  MoveC 574 to (267.87, -55.04, -8.35) mm, rotated rx -180 ry 0 rz 0 deg; joints [19.602, -53.093, 148.442, 19.65, -94.169, 2.069] to (268.06, -55.49, -8.35) mm, rotated rx 180 ry 0 rz 0 deg; joints [19.58, -53.096, 148.465, 19.628, -94.189, 2.074]
  MoveL 575 to (268.06, -80.89, -8.35) mm, rotated rx 180 ry 0 rz 0 deg; joints [18.089, -53.148, 149.041, 18.147, -94.732, 2.105]
  MoveL 576 to (217.26, -80.89, -8.35) mm, rotated rx -180 ry 0 rz 0 deg; joints [17.156, -52.603, 145.594, 17.161, -91.988, 1.155]
  MoveL 577 to (217.26, -30.09, -8.35) mm, rotated rx -180 ry 0 rz 0 deg; joints [19.982, -52.424, 144.438, 19.979, -91.023, 0.96]
  MoveL 578 to (268.06, -30.09, -8.35) mm, rotated rx -180 ry 0 rz 0 deg; joints [21.044, -53.031, 147.845, 21.081, -93.623, 2.002]
  MoveL 579 to (268.06, -55.49, -8.35) mm, rotated rx 180 ry 0 rz 0 deg; joints [19.58, -53.096, 148.465, 19.628, -94.189, 2.074]
  MoveC 580 to (267.87, -55.94, -8.35) mm, rotated rx -180 ry 0 rz 0 deg; joints [19.55, -53.095, 148.464, 19.598, -94.189, 2.071] to (267.42, -56.12, -8.35) mm, rotated rx 180 ry 0 rz 0 deg; joints [19.53, -53.092, 148.438, 19.578, -94.169, 2.062]
  MoveL 581 to (266.79, -56.12, -8.35) mm, rotated rx 180 ry 0 rz 0 deg; joints [19.517, -53.086, 148.396, 19.564, -94.135, 2.048]
  MoveC 582 to (266.34, -56.12, -8.16) mm, rotated rx 180 ry 0 rz 0 deg; joints [19.508, -53.1, 148.369, 19.553, -94.096, 2.034] to (266.15, -56.12, -7.72) mm, rotated rx 180 ry 0 rz 0 deg; joints [19.504, -53.144, 148.364, 19.548, -94.051, 2.017]
  Set speed (1000.0 mm/s)
  MoveL 583 to (266.15, -56.12, 6) mm, rotated rx 180 ry 0 rz 0 deg; joints [19.495, -54.53, 148.591, 19.516, -92.959, 1.628]
  MoveL 584 to (139.15, -54.85, 6) mm, rotated rx 180 ry 0 rz 0 deg; joints [17.25, -52.506, 139.813, 17.276, -86.559, -0.527]
  Set speed (25.4 mm/s)
  MoveL 585 to (139.15, -54.85, -3.54) mm, rotated rx -180 ry 0 rz 0 deg; joints [17.254, -51.692, 139.679, 17.269, -87.209, -0.325]
  MoveC 586 to (139.34, -54.85, -3.99) mm, rotated rx 180 ry 0 rz 0 deg; joints [17.258, -51.657, 139.686, 17.272, -87.248, -0.313] to (139.79, -54.85, -4.17) mm, rotated rx 180 ry 0 rz 0 deg; joints [17.265, -51.649, 139.715, 17.279, -87.283, -0.302]
  Set speed (50.8 mm/s)
  MoveL 587 to (140.42, -54.85, -4.18) mm, rotated rx 180 ry 0 rz 0 deg; joints [17.275, -51.661, 139.76, 17.289, -87.315, -0.293]
  MoveC 588 to (140.87, -55.04, -4.17) mm, rotated rx -180 ry 0 rz 0 deg; joints [17.273, -51.67, 139.795, 17.286, -87.34, -0.285] to (141.06, -55.49, -4.17) mm, rotated rx -180 ry 0 rz 0 deg; joints [17.252, -51.676, 139.818, 17.265, -87.356, -0.279]
  MoveL 589 to (141.06, -80.89, -4.18) mm, rotated rx -180 ry 0 rz 0 deg; joints [15.918, -51.795, 140.349, 15.924, -87.74, -0.124]
  MoveL 590 to (90.26, -80.89, -4.17) mm, rotated rx 180 ry 0 rz 0 deg; joints [15.186, -50.797, 136.713, 15.235, -85.19, -0.8]
  MoveL 591 to (90.26, -30.09, -4.17) mm, rotated rx 180 ry 0 rz 0 deg; joints [17.729, -50.515, 135.638, 17.808, -84.486, -1.218]
  MoveL 592 to (141.06, -30.09, -4.17) mm, rotated rx -180 ry 0 rz 0 deg; joints [18.568, -51.543, 139.244, 18.589, -86.951, -0.46]
  MoveL 593 to (141.06, -55.49, -4.17) mm, rotated rx -180 ry 0 rz 0 deg; joints [17.252, -51.676, 139.818, 17.265, -87.356, -0.279]
  MoveC 594 to (140.87, -55.94, -4.18) mm, rotated rx 180 ry 0 rz 0 deg; joints [17.226, -51.675, 139.815, 17.239, -87.354, -0.279] to (140.42, -56.12, -4.17) mm, rotated rx -180 ry 0 rz 0 deg; joints [17.209, -51.668, 139.787, 17.222, -87.334, -0.284]
  MoveL 595 to (139.79, -56.12, -4.18) mm, rotated rx -180 ry 0 rz 0 deg; joints [17.199, -51.656, 139.742, 17.212, -87.303, -0.294]
  MoveC 596 to (139.34, -56.12, -3.99) mm, rotated rx -180 ry 0 rz 0 deg; joints [17.192, -51.663, 139.713, 17.205, -87.268, -0.304] to (139.15, -56.12, -3.54) mm, rotated rx -180 ry 0 rz 0 deg; joints [17.188, -51.698, 139.707, 17.203, -87.228, -0.317]
  Set speed (1000.0 mm/s)
  MoveL 597 to (139.15, -56.12, 5) mm, rotated rx 180 ry 0 rz 0 deg; joints [17.184, -52.427, 139.827, 17.208, -86.647, -0.497]
  MoveL 598 to (139.15, -54.85, 5) mm, rotated rx -180 ry 0 rz 0 deg; joints [17.25, -52.421, 139.8, 17.275, -86.628, -0.506]
  Set speed (25.4 mm/s)
  MoveL 599 to (139.15, -54.85, 1.83) mm, rotated rx -180 ry 0 rz 0 deg; joints [17.252, -52.15, 139.756, 17.273, -86.844, -0.438]
  MoveL 600 to (139.15, -54.85, -7.72) mm, rotated rx -180 ry 0 rz 0 deg; joints [17.257, -51.335, 139.618, 17.267, -87.49, -0.237]
  MoveC 601 to (139.34, -54.85, -8.16) mm, rotated rx -180 ry 0 rz 0 deg; joints [17.26, -51.3, 139.624, 17.27, -87.53, -0.225] to (139.79, -54.85, -8.35) mm, rotated rx -180 ry 0 rz 0 deg; joints [17.267, -51.293, 139.653, 17.277, -87.565, -0.215]
  Set speed (50.8 mm/s)
  MoveL 602 to (140.42, -54.85, -8.35) mm, rotated rx 180 ry 0 rz 0 deg; joints [17.277, -51.304, 139.698, 17.287, -87.596, -0.205]
  MoveC 603 to (140.87, -55.04, -8.35) mm, rotated rx 180 ry 0 rz 0 deg; joints [17.275, -51.313, 139.733, 17.284, -87.622, -0.197] to (141.06, -55.49, -8.35) mm, rotated rx -180 ry 0 rz 0 deg; joints [17.255, -51.319, 139.756, 17.264, -87.638, -0.191]
  MoveL 604 to (141.06, -80.89, -8.35) mm, rotated rx 180 ry 0 rz 0 deg; joints [15.92, -51.434, 140.287, 15.923, -88.027, -0.043]
  MoveL 605 to (90.26, -80.89, -8.35) mm, rotated rx -180 ry 0 rz 0 deg; joints [15.188, -50.458, 136.654, 15.231, -85.46, -0.726]
  MoveL 606 to (90.26, -30.09, -8.35) mm, rotated rx -180 ry 0 rz 0 deg; joints [17.731, -50.182, 135.58, 17.802, -84.747, -1.134]
  MoveL 607 to (141.06, -30.09, -8.35) mm, rotated rx 180 ry 0 rz 0 deg; joints [18.57, -51.189, 139.183, 18.587, -87.228, -0.367]
  MoveL 608 to (141.06, -55.49, -8.35) mm, rotated rx -180 ry 0 rz 0 deg; joints [17.255, -51.319, 139.756, 17.264, -87.638, -0.191]
  MoveC 609 to (140.87, -55.94, -8.35) mm, rotated rx 180 ry 0 rz 0 deg; joints [17.228, -51.318, 139.753, 17.237, -87.636, -0.191] to (140.42, -56.12, -8.35) mm, rotated rx 180 ry 0 rz 0 deg; joints [17.211, -51.31, 139.725, 17.22, -87.616, -0.197]
  MoveL 610 to (139.79, -56.12, -8.35) mm, rotated rx 180 ry 0 rz 0 deg; joints [17.201, -51.299, 139.681, 17.21, -87.585, -0.206]
  MoveC 611 to (139.34, -56.12, -8.16) mm, rotated rx -180 ry 0 rz 0 deg; joints [17.194, -51.306, 139.652, 17.204, -87.55, -0.217] to (139.15, -56.12, -7.72) mm, rotated rx 180 ry 0 rz 0 deg; joints [17.19, -51.341, 139.645, 17.201, -87.51, -0.229]
  Set speed (1000.0 mm/s)
  MoveL 612 to (139.15, -56.12, 6) mm, rotated rx -180 ry 0 rz 0 deg; joints [17.184, -52.513, 139.841, 17.209, -86.578, -0.518]
  MoveL 613 to (139.15, -235.88, 6) mm, rotated rx -180 ry 0 rz 0 deg; joints [7.413, -53.13, 142.645, 7.41, -88.649, 0.21]
  Set speed (25.4 mm/s)
  MoveL 614 to (139.15, -235.88, -3.54) mm, rotated rx -180 ry 0 rz 0 deg; joints [7.416, -52.274, 142.505, 7.412, -89.36, 0.302]
  MoveC 615 to (139.34, -235.88, -3.99) mm, rotated rx -180 ry 0 rz 0 deg; joints [7.418, -52.236, 142.511, 7.413, -89.403, 0.308] to (139.79, -235.88, -4.17) mm, rotated rx -180 ry 0 rz 0 deg; joints [7.421, -52.227, 142.541, 7.416, -89.442, 0.313]
  Set speed (50.8 mm/s)
  MoveL 616 to (140.42, -235.88, -4.18) mm, rotated rx -180 ry 0 rz 0 deg; joints [7.426, -52.238, 142.587, 7.421, -89.477, 0.317]
  MoveC 617 to (140.87, -236.07, -4.18) mm, rotated rx -180 ry 0 rz 0 deg; joints [7.419, -52.245, 142.621, 7.414, -89.503, 0.321] to (141.06, -236.52, -4.17) mm, rotated rx -180 ry 0 rz 0 deg; joints [7.395, -52.249, 142.639, 7.39, -89.517, 0.322]
  MoveL 618 to (141.06, -261.92, -4.18) mm, rotated rx 180 ry 0 rz 0 deg; joints [5.961, -52.283, 142.851, 5.956, -89.695, 0.331]
  MoveL 619 to (90.26, -261.92, -4.17) mm, rotated rx -180 ry 0 rz 0 deg; joints [5.676, -51.366, 139.142, 5.679, -86.918, 0.052]
  MoveL 620 to (90.26, -211.12, -4.18) mm, rotated rx -180 ry 0 rz 0 deg; joints [8.4, -51.27, 138.686, 8.41, -86.574, -0.106]
  MoveL 621 to (141.06, -211.12, -4.17) mm, rotated rx -180 ry 0 rz 0 deg; joints [8.819, -52.205, 142.38, 8.814, -89.304, 0.299]
  MoveL 622 to (141.06, -236.52, -4.17) mm, rotated rx -180 ry 0 rz 0 deg; joints [7.395, -52.249, 142.639, 7.39, -89.517, 0.322]
  MoveC 623 to (140.87, -236.97, -4.17) mm, rotated rx -180 ry 0 rz 0 deg; joints [7.368, -52.247, 142.629, 7.363, -89.51, 0.321] to (140.42, -237.15, -4.18) mm, rotated rx -180 ry 0 rz 0 deg; joints [7.354, -52.24, 142.599, 7.35, -89.486, 0.318]
  MoveL 624 to (139.79, -237.16, -4.17) mm, rotated rx 180 ry 0 rz 0 deg; joints [7.35, -52.229, 142.553, 7.345, -89.451, 0.314]
  MoveC 625 to (139.34, -237.16, -3.99) mm, rotated rx 180 ry 0 rz 0 deg; joints [7.346, -52.238, 142.523, 7.342, -89.413, 0.309] to (139.15, -237.15, -3.54) mm, rotated rx 180 ry 0 rz 0 deg; joints [7.345, -52.276, 142.517, 7.34, -89.369, 0.303]
  Set speed (1000.0 mm/s)
  MoveL 626 to (139.15, -237.15, 5) mm, rotated rx -180 ry 0 rz 0 deg; joints [7.342, -53.043, 142.643, 7.338, -88.734, 0.221]
  MoveL 627 to (139.15, -235.88, 5) mm, rotated rx 180 ry 0 rz 0 deg; joints [7.413, -53.041, 142.631, 7.41, -88.724, 0.219]
  Set speed (25.4 mm/s)
  MoveL 628 to (139.15, -235.88, 1.83) mm, rotated rx -180 ry 0 rz 0 deg; joints [7.414, -52.755, 142.585, 7.41, -88.961, 0.25]
  MoveL 629 to (139.15, -235.89, -7.72) mm, rotated rx -180 ry 0 rz 0 deg; joints [7.418, -51.899, 142.44, 7.413, -89.668, 0.342]
  MoveC 630 to (139.34, -235.88, -8.16) mm, rotated rx -180 ry 0 rz 0 deg; joints [7.419, -51.861, 142.447, 7.414, -89.711, 0.348] to (139.79, -235.88, -8.35) mm, rotated rx -180 ry 0 rz 0 deg; joints [7.423, -51.852, 142.476, 7.418, -89.75, 0.353]
  Set speed (50.8 mm/s)
  MoveL 631 to (140.42, -235.88, -8.35) mm, rotated rx -180 ry 0 rz 0 deg; joints [7.427, -51.862, 142.522, 7.422, -89.785, 0.358]
  MoveC 632 to (140.87, -236.07, -8.35) mm, rotated rx -180 ry 0 rz 0 deg; joints [7.42, -51.87, 142.556, 7.415, -89.811, 0.361] to (141.06, -236.52, -8.35) mm, rotated rx 180 ry 0 rz 0 deg; joints [7.396, -51.873, 142.574, 7.391, -89.825, 0.362]
  MoveL 633 to (141.06, -261.92, -8.35) mm, rotated rx 180 ry 0 rz 0 deg; joints [5.963, -51.906, 142.786, 5.958, -90.006, 0.364]
  MoveL 634 to (90.26, -261.92, -8.35) mm, rotated rx 180 ry 0 rz 0 deg; joints [5.677, -51.013, 139.081, 5.679, -87.208, 0.081]
  MoveL 635 to (90.26, -211.12, -8.35) mm, rotated rx -180 ry 0 rz 0 deg; joints [8.401, -50.92, 138.625, 8.409, -86.86, -0.063]
  MoveL 636 to (141.06, -211.12, -8.35) mm, rotated rx -180 ry 0 rz 0 deg; joints [8.821, -51.83, 142.316, 8.816, -89.61, 0.347]
  MoveL 637 to (141.06, -236.52, -8.35) mm, rotated rx 180 ry 0 rz 0 deg; joints [7.396, -51.873, 142.574, 7.391, -89.825, 0.362]
  MoveC 638 to (140.87, -236.97, -8.35) mm, rotated rx -180 ry 0 rz 0 deg; joints [7.37, -51.871, 142.564, 7.365, -89.818, 0.361] to (140.42, -237.16, -8.35) mm, rotated rx 180 ry 0 rz 0 deg; joints [7.356, -51.864, 142.534, 7.351, -89.795, 0.358]
  MoveL 639 to (139.79, -237.16, -8.35) mm, rotated rx -180 ry 0 rz 0 deg; joints [7.351, -51.854, 142.488, 7.346, -89.759, 0.353]
  MoveC 640 to (139.34, -237.15, -8.16) mm, rotated rx -180 ry 0 rz 0 deg; joints [7.348, -51.863, 142.458, 7.343, -89.721, 0.348] to (139.15, -237.15, -7.72) mm, rotated rx -180 ry 0 rz 0 deg; joints [7.346, -51.9, 142.452, 7.342, -89.678, 0.343]
  Set speed (1000.0 mm/s)
  MoveL 641 to (139.15, -237.15, 6) mm, rotated rx 180 ry 0 rz 0 deg; joints [7.341, -53.133, 142.657, 7.338, -88.659, 0.212]
  MoveL 642 to (266.15, -235.89, 6) mm, rotated rx -180 ry 0 rz 0 deg; joints [8.471, -54.806, 151.649, 8.512, -95.899, 1.283]
  Set speed (25.4 mm/s)
  MoveL 643 to (266.15, -235.89, -3.54) mm, rotated rx 180 ry 0 rz 0 deg; joints [8.476, -53.774, 151.483, 8.53, -96.755, 1.413]
  MoveC 644 to (266.34, -235.89, -3.99) mm, rotated rx -180 ry 0 rz 0 deg; joints [8.478, -53.727, 151.487, 8.533, -96.806, 1.421] to (266.79, -235.88, -4.17) mm, rotated rx -180 ry 0 rz 0 deg; joints [8.482, -53.709, 151.515, 8.538, -96.851, 1.428]
  Set speed (50.8 mm/s)
  MoveL 645 to (267.42, -235.89, -4.17) mm, rotated rx 180 ry 0 rz 0 deg; joints [8.488, -53.713, 151.559, 8.545, -96.89, 1.435]
  MoveC 646 to (267.87, -236.07, -4.18) mm, rotated rx 180 ry 0 rz 0 deg; joints [8.48, -53.715, 151.592, 8.538, -96.921, 1.438] to (268.06, -236.52, -4.17) mm, rotated rx -180 ry 0 rz 0 deg; joints [8.453, -53.716, 151.609, 8.511, -96.937, 1.437]
  MoveL 647 to (268.06, -261.92, -4.18) mm, rotated rx -180 ry 0 rz 0 deg; joints [6.819, -53.716, 151.842, 6.868, -97.198, 1.241]
  MoveL 648 to (217.26, -261.92, -4.18) mm, rotated rx 180 ry 0 rz 0 deg; joints [6.448, -53.314, 148.292, 6.459, -94.076, 0.832]
  MoveL 649 to (217.26, -211.12, -4.18) mm, rotated rx 180 ry 0 rz 0 deg; joints [9.532, -53.273, 147.796, 9.546, -93.591, 1.022]
  MoveL 650 to (268.06, -211.12, -4.17) mm, rotated rx -180 ry 0 rz 0 deg; joints [10.074, -53.712, 151.327, 10.138, -96.628, 1.609]
  MoveL 651 to (268.06, -236.52, -4.17) mm, rotated rx -180 ry 0 rz 0 deg; joints [8.453, -53.716, 151.609, 8.511, -96.937, 1.437]
  MoveC 652 to (267.87, -236.97, -4.17) mm, rotated rx -180 ry 0 rz 0 deg; joints [8.423, -53.715, 151.601, 8.48, -96.931, 1.432] to (267.42, -237.16, -4.17) mm, rotated rx -180 ry 0 rz 0 deg; joints [8.407, -53.713, 151.572, 8.463, -96.905, 1.426]
  MoveL 653 to (266.79, -237.15, -4.18) mm, rotated rx -180 ry 0 rz 0 deg; joints [8.401, -53.709, 151.528, 8.457, -96.865, 1.419]
  MoveC 654 to (266.34, -237.15, -3.99) mm, rotated rx -180 ry 0 rz 0 deg; joints [8.396, -53.727, 151.5, 8.451, -96.82, 1.412] to (266.15, -237.16, -3.54) mm, rotated rx -180 ry 0 rz 0 deg; joints [8.394, -53.774, 151.495, 8.449, -96.769, 1.404]
  Set speed (1000.0 mm/s)
  MoveL 655 to (266.15, -237.15, 5) mm, rotated rx 180 ry 0 rz 0 deg; joints [8.391, -54.698, 151.645, 8.432, -96.003, 1.289]
  MoveL 656 to (266.15, -235.89, 5) mm, rotated rx -180 ry 0 rz 0 deg; joints [8.472, -54.698, 151.632, 8.513, -95.989, 1.297]
  Set speed (25.4 mm/s)
  MoveL 657 to (266.15, -235.89, 1.83) mm, rotated rx -180 ry 0 rz 0 deg; joints [8.473, -54.354, 151.577, 8.52, -96.275, 1.34]
  MoveL 658 to (266.15, -235.89, -7.71) mm, rotated rx -180 ry 0 rz 0 deg; joints [8.477, -53.323, 151.406, 8.539, -97.125, 1.469]
  MoveC 659 to (266.34, -235.88, -8.16) mm, rotated rx -180 ry 0 rz 0 deg; joints [8.479, -53.276, 151.411, 8.542, -97.176, 1.477] to (266.79, -235.89, -8.35) mm, rotated rx -180 ry 0 rz 0 deg; joints [8.484, -53.258, 151.438, 8.547, -97.221, 1.484]
  Set speed (50.8 mm/s)
  MoveL 660 to (267.42, -235.89, -8.35) mm, rotated rx -180 ry 0 rz 0 deg; joints [8.49, -53.261, 151.482, 8.554, -97.261, 1.491]
  MoveC 661 to (267.87, -236.07, -8.35) mm, rotated rx 180 ry 0 rz 0 deg; joints [8.482, -53.264, 151.515, 8.547, -97.291, 1.495] to (268.06, -236.52, -8.35) mm, rotated rx -180 ry 0 rz 0 deg; joints [8.455, -53.264, 151.532, 8.52, -97.308, 1.493]
  MoveL 662 to (268.06, -261.92, -8.35) mm, rotated rx -180 ry 0 rz 0 deg; joints [6.82, -53.262, 151.764, 6.876, -97.573, 1.287]
  MoveL 663 to (217.26, -261.92, -8.35) mm, rotated rx 180 ry 0 rz 0 deg; joints [6.449, -52.894, 148.22, 6.464, -94.423, 0.871]
  MoveL 664 to (217.26, -211.12, -8.35) mm, rotated rx 180 ry 0 rz 0 deg; joints [9.534, -52.857, 147.725, 9.551, -93.931, 1.079]
  MoveL 665 to (268.06, -211.12, -8.35) mm, rotated rx -180 ry 0 rz 0 deg; joints [10.076, -53.263, 151.251, 10.147, -96.995, 1.675]
  MoveL 666 to (268.06, -236.52, -8.35) mm, rotated rx 180 ry 0 rz 0 deg; joints [8.455, -53.264, 151.532, 8.52, -97.308, 1.493]
  MoveC 667 to (267.87, -236.97, -8.35) mm, rotated rx -180 ry 0 rz 0 deg; joints [8.425, -53.264, 151.524, 8.489, -97.302, 1.488] to (267.42, -237.16, -8.35) mm, rotated rx 180 ry 0 rz 0 deg; joints [8.409, -53.261, 151.495, 8.472, -97.275, 1.481]
  MoveL 668 to (266.79, -237.16, -8.35) mm, rotated rx 180 ry 0 rz 0 deg; joints [8.403, -53.258, 151.451, 8.465, -97.235, 1.475]
  MoveC 669 to (266.34, -237.16, -8.16) mm, rotated rx -180 ry 0 rz 0 deg; joints [8.398, -53.276, 151.424, 8.46, -97.191, 1.467] to (266.15, -237.16, -7.72) mm, rotated rx 180 ry 0 rz 0 deg; joints [8.396, -53.323, 151.419, 8.457, -97.139, 1.459]
  Set speed (1000.0 mm/s)
  MoveL 670 to (266.15, -237.16, 6) mm, rotated rx 180 ry 0 rz 0 deg; joints [8.39, -54.806, 151.662, 8.43, -95.912, 1.275]
  MoveL 671 to (393.15, -235.88, 6) mm, rotated rx -180 ry 0 rz -30 deg; joints [-2.482, -54.877, 157.892, -33.089, -100.339, -6.392]
  Set speed (25.4 mm/s)
  MoveL 672 to (393.15, -235.89, -3.54) mm, rotated rx 180 ry 0 rz -30 deg; joints [-2.479, -53.673, 157.698, -33.192, -101.185, -6.954]
  MoveC 673 to (393.34, -235.88, -3.99) mm, rotated rx 180 ry 0 rz -30 deg; joints [-2.479, -53.615, 157.701, -33.199, -101.236, -6.988] to (393.79, -235.89, -4.18) mm, rotated rx 180 ry 0 rz -30 deg; joints [-2.481, -53.588, 157.727, -33.206, -101.28, -7.018]
  Set speed (50.8 mm/s)
  MoveL 674 to (394.42, -235.88, -4.18) mm, rotated rx -180 ry 0 rz -30 deg; joints [-2.483, -53.584, 157.77, -33.213, -101.319, -7.045]
  MoveC 675 to (394.87, -236.07, -4.18) mm, rotated rx 180 ry 0 rz -30 deg; joints [-2.498, -53.58, 157.8, -33.232, -101.345, -7.066] to (395.06, -236.52, -4.17) mm, rotated rx -180 ry 0 rz -30 deg; joints [-2.531, -53.579, 157.811, -33.266, -101.351, -7.08]
  MoveL 676 to (395.06, -261.92, -4.17) mm, rotated rx -180 ry 0 rz -30 deg; joints [-4.359, -53.578, 157.706, -35.101, -101.013, -7.398]
  MoveL 677 to (344.26, -261.92, -4.18) mm, rotated rx -180 ry 0 rz -30 deg; joints [-4.098, -53.729, 154.244, -34.491, -98.078, -5.261]
  MoveL 678 to (344.26, -211.12, -4.17) mm, rotated rx -180 ry 0 rz 0 deg; joints [11.013, -53.827, 156.503, 11.239, -101.571, 2.724]
  MoveL 679 to (395.06, -211.12, -4.18) mm, rotated rx -180 ry 0 rz 30 deg; joints [22.093, -54.031, 153.781, 52.376, -95.091, 7.51]
  MoveL 680 to (395.06, -236.52, -4.18) mm, rotated rx -180 ry 0 rz 30 deg; joints [20.495, -54.016, 154.413, 50.834, -95.712, 7.845]
  MoveC 681 to (394.87, -236.97, -4.17) mm, rotated rx -180 ry 0 rz 30 deg; joints [20.462, -54.015, 154.412, 50.802, -95.716, 7.841] to (394.42, -237.15, -4.18) mm, rotated rx -180 ry 0 rz 30 deg; joints [20.44, -54.015, 154.387, 50.777, -95.704, 7.82]
  MoveL 682 to (393.79, -237.15, -4.18) mm, rotated rx -180 ry 0 rz 30 deg; joints [20.425, -54.014, 154.346, 50.759, -95.681, 7.787]
  MoveC 683 to (393.34, -237.16, -3.99) mm, rotated rx 180 ry 0 rz 30 deg; joints [20.414, -54.035, 154.321, 50.745, -95.653, 7.749] to (393.15, -237.16, -3.54) mm, rotated rx 180 ry 0 rz 30 deg; joints [20.409, -54.086, 154.317, 50.736, -95.619, 7.706]
  Set speed (1000.0 mm/s)
  MoveL 684 to (393.15, -237.16, 5) mm, rotated rx -180 ry 0 rz 30 deg; joints [20.404, -55.074, 154.476, 50.67, -95.094, 7.061]
  MoveL 685 to (393.15, -235.88, 5) mm, rotated rx -180 ry 0 rz 30 deg; joints [20.484, -55.075, 154.445, 50.748, -95.065, 7.045]
  Set speed (25.4 mm/s)
  MoveL 686 to (393.15, -235.88, 1.82) mm, rotated rx 180 ry 0 rz 30 deg; joints [20.486, -54.707, 154.388, 50.772, -95.26, 7.286]
  MoveL 687 to (393.15, -235.88, -7.72) mm, rotated rx -180 ry 0 rz 30 deg; joints [20.493, -53.606, 154.206, 50.848, -95.84, 8.003]
  MoveC 688 to (393.34, -235.89, -8.16) mm, rotated rx -180 ry 0 rz 30 deg; joints [20.497, -53.554, 154.209, 50.857, -95.874, 8.046] to (393.79, -235.88, -8.35) mm, rotated rx 180 ry 0 rz 30 deg; joints [20.508, -53.533, 154.234, 50.871, -95.902, 8.084]
  Set speed (50.8 mm/s)
  MoveL 689 to (394.42, -235.89, -8.35) mm, rotated rx -180 ry 0 rz 30 deg; joints [20.523, -53.534, 154.275, 50.889, -95.925, 8.117]
  MoveC 690 to (394.87, -236.07, -8.35) mm, rotated rx -180 ry 0 rz 30 deg; joints [20.522, -53.534, 154.309, 50.891, -95.947, 8.143] to (395.06, -236.52, -8.35) mm, rotated rx -180 ry 0 rz 30 deg; joints [20.498, -53.533, 154.331, 50.869, -95.965, 8.158]
  MoveL 691 to (395.06, -261.92, -8.35) mm, rotated rx -180 ry 0 rz 30 deg; joints [18.866, -53.5, 154.914, 49.297, -96.601, 8.431]
  MoveL 692 to (344.26, -261.92, -8.35) mm, rotated rx 180 ry 0 rz 0 deg; joints [7.464, -53.229, 156.963, 7.649, -102.746, 2.083]
  MoveL 693 to (344.26, -211.12, -8.35) mm, rotated rx 180 ry 0 rz 0 deg; joints [11.015, -53.318, 156.416, 11.258, -101.985, 2.809]
  MoveL 694 to (395.06, -211.12, -8.35) mm, rotated rx -180 ry 0 rz 30 deg; joints [22.096, -53.555, 153.7, 52.407, -95.332, 7.825]
  MoveL 695 to (395.06, -236.52, -8.35) mm, rotated rx -180 ry 0 rz 30 deg; joints [20.498, -53.533, 154.331, 50.869, -95.965, 8.158]
  MoveC 696 to (394.87, -236.97, -8.35) mm, rotated rx 180 ry 0 rz 30 deg; joints [20.465, -53.533, 154.33, 50.836, -95.969, 8.154] to (394.42, -237.16, -8.35) mm, rotated rx -180 ry 0 rz 30 deg; joints [20.443, -53.532, 154.306, 50.812, -95.957, 8.132]
  MoveL 697 to (393.79, -237.15, -8.35) mm, rotated rx -180 ry 0 rz 30 deg; joints [20.428, -53.532, 154.265, 50.794, -95.934, 8.099]
  MoveC 698 to (393.34, -237.16, -8.16) mm, rotated rx 180 ry 0 rz 30 deg; joints [20.417, -53.553, 154.239, 50.779, -95.906, 8.061] to (393.15, -237.16, -7.72) mm, rotated rx -180 ry 0 rz 30 deg; joints [20.412, -53.605, 154.236, 50.77, -95.872, 8.018]
  Set speed (1000.0 mm/s)
  MoveL 699 to (393.15, -237.15, 6) mm, rotated rx -180 ry 0 rz 30 deg; joints [20.403, -55.19, 154.494, 50.663, -95.032, 6.985]
  MoveL 700 to (393.15, -422.22, 6) mm, rotated rx -180 ry 0 rz 30 deg; joints [7.885, -54.996, 157.593, 38.441, -99.031, 7.595]
  Set speed (25.4 mm/s)
  MoveL 701 to (393.15, -422.22, -3.54) mm, rotated rx -180 ry 0 rz 30 deg; joints [7.89, -53.801, 157.401, 38.549, -99.815, 8.228]
  MoveC 702 to (393.34, -422.22, -3.99) mm, rotated rx -180 ry 0 rz 30 deg; joints [7.892, -53.744, 157.404, 38.557, -99.862, 8.267] to (393.79, -422.22, -4.17) mm, rotated rx 180 ry 0 rz 30 deg; joints [7.896, -53.718, 157.43, 38.568, -99.902, 8.301]
  Set speed (50.8 mm/s)
  MoveL 703 to (394.42, -422.22, -4.18) mm, rotated rx -180 ry 0 rz 30 deg; joints [7.902, -53.714, 157.473, 38.579, -99.938, 8.331]
  MoveC 704 to (394.87, -422.41, -4.18) mm, rotated rx -180 ry 0 rz 30 deg; joints [7.894, -53.711, 157.505, 38.574, -99.966, 8.352] to (395.06, -422.86, -4.18) mm, rotated rx -180 ry 0 rz 30 deg; joints [7.863, -53.709, 157.522, 38.546, -99.985, 8.358]
  MoveL 705 to (395.06, -448.26, -4.17) mm, rotated rx -180 ry 0 rz 30 deg; joints [6.05, -53.668, 157.726, 36.75, -100.447, 8.159]
  MoveL 706 to (344.26, -448.26, -4.18) mm, rotated rx 180 ry 0 rz 30 deg; joints [5.687, -53.812, 154.272, 36.047, -97.596, 5.935]
  MoveL 707 to (344.26, -397.46, -4.18) mm, rotated rx 180 ry 0 rz 0 deg; joints [-2.223, -53.617, 157.457, -2.285, -102.959, -0.274]
  MoveL 708 to (395.06, -397.46, -4.18) mm, rotated rx -180 ry 0 rz -30 deg; joints [-13.884, -53.653, 156.233, -44.491, -98.421, -8.11]
  MoveL 709 to (395.06, -422.86, -4.17) mm, rotated rx 180 ry 0 rz -30 deg; joints [-15.601, -53.67, 155.791, -46.158, -97.837, -8.041]
  MoveC 710 to (394.87, -423.31, -4.18) mm, rotated rx -180 ry 0 rz -30 deg; joints [-15.628, -53.671, 155.77, -46.182, -97.819, -8.029] to (394.42, -423.49, -4.18) mm, rotated rx -180 ry 0 rz -30 deg; joints [-15.632, -53.672, 155.737, -46.183, -97.794, -8.005]
  MoveL 711 to (393.79, -423.49, -4.17) mm, rotated rx -180 ry 0 rz -30 deg; joints [-15.62, -53.673, 155.695, -46.167, -97.766, -7.971]
  MoveC 712 to (393.34, -423.49, -3.99) mm, rotated rx 180 ry 0 rz -30 deg; joints [-15.611, -53.696, 155.67, -46.153, -97.733, -7.935] to (393.15, -423.49, -3.54) mm, rotated rx -180 ry 0 rz -30 deg; joints [-15.608, -53.75, 155.666, -46.144, -97.694, -7.892]
  Set speed (1000.0 mm/s)
  MoveL 713 to (393.15, -423.49, 5) mm, rotated rx 180 ry 0 rz -30 deg; joints [-15.608, -54.772, 155.832, -46.065, -97.1, -7.27]
  MoveL 714 to (393.15, -422.22, 5) mm, rotated rx 180 ry 0 rz -30 deg; joints [-15.523, -54.772, 155.855, -45.982, -97.128, -7.276]
  Set speed (25.4 mm/s)
  MoveL 715 to (393.15, -422.22, 1.82) mm, rotated rx -180 ry 0 rz -30 deg; joints [-15.523, -54.392, 155.795, -46.011, -97.351, -7.508]
  MoveL 716 to (393.15, -422.22, -7.71) mm, rotated rx -180 ry 0 rz -30 deg; joints [-15.523, -53.251, 155.605, -46.103, -98.011, -8.198]
  MoveC 717 to (393.34, -422.22, -8.16) mm, rotated rx 180 ry 0 rz -30 deg; joints [-15.526, -53.197, 155.608, -46.112, -98.05, -8.24] to (393.79, -422.22, -8.35) mm, rotated rx -180 ry 0 rz -30 deg; joints [-15.534, -53.174, 155.634, -46.126, -98.082, -8.277]
  Set speed (50.8 mm/s)
  MoveL 718 to (394.42, -422.22, -8.35) mm, rotated rx 180 ry 0 rz -30 deg; joints [-15.546, -53.172, 155.676, -46.142, -98.111, -8.311]
  MoveC 719 to (394.87, -422.41, -8.35) mm, rotated rx 180 ry 0 rz -30 deg; joints [-15.567, -53.171, 155.702, -46.165, -98.127, -8.334] to (395.06, -422.86, -8.35) mm, rotated rx 180 ry 0 rz -30 deg; joints [-15.601, -53.17, 155.706, -46.199, -98.124, -8.342]
  MoveL 720 to (395.06, -448.26, -8.35) mm, rotated rx -180 ry 0 rz -30 deg; joints [-17.289, -53.19, 155.214, -47.832, -97.513, -8.212]
  MoveL 721 to (344.26, -448.26, -8.35) mm, rotated rx 180 ry 0 rz 0 deg; joints [-5.849, -53.098, 157.121, -6.009, -103.08, -1.181]
  MoveL 722 to (344.26, -397.46, -8.35) mm, rotated rx -180 ry 0 rz 0 deg; joints [-2.222, -53.096, 157.368, -2.288, -103.392, -0.292]
  MoveL 723 to (395.06, -397.46, -8.35) mm, rotated rx 180 ry 0 rz -30 deg; joints [-13.884, -53.148, 156.147, -44.535, -98.72, -8.407]
  MoveL 724 to (395.06, -422.86, -8.35) mm, rotated rx 180 ry 0 rz -30 deg; joints [-15.601, -53.17, 155.706, -46.199, -98.124, -8.342]
  MoveC 725 to (394.87, -423.31, -8.35) mm, rotated rx -180 ry 0 rz -30 deg; joints [-15.627, -53.171, 155.685, -46.224, -98.105, -8.331] to (394.42, -423.49, -8.35) mm, rotated rx -180 ry 0 rz -30 deg; joints [-15.631, -53.173, 155.652, -46.224, -98.081, -8.306]
  MoveL 726 to (393.79, -423.49, -8.35) mm, rotated rx -180 ry 0 rz -30 deg; joints [-15.62, -53.175, 155.61, -46.208, -98.052, -8.273]
  MoveC 727 to (393.34, -423.49, -8.16) mm, rotated rx 180 ry 0 rz -30 deg; joints [-15.611, -53.198, 155.585, -46.195, -98.02, -8.235] to (393.15, -423.49, -7.72) mm, rotated rx -180 ry 0 rz -30 deg; joints [-15.608, -53.252, 155.582, -46.185, -97.981, -8.193]
  Set speed (1000.0 mm/s)
  MoveL 728 to (393.15, -423.49, 6) mm, rotated rx -180 ry 0 rz -30 deg; joints [-15.608, -54.892, 155.851, -46.056, -97.03, -7.197]
  MoveL 729 to (266.15, -422.22, 6) mm, rotated rx 180 ry 0 rz 0 deg; joints [-3.642, -54.753, 152.184, -3.67, -96.547, -0.202]
  Set speed (25.4 mm/s)
  MoveL 730 to (266.15, -422.22, -3.54) mm, rotated rx 180 ry 0 rz 0 deg; joints [-3.64, -53.708, 152.015, -3.674, -97.421, -0.258]
  MoveC 731 to (266.34, -422.22, -3.99) mm, rotated rx 180 ry 0 rz 0 deg; joints [-3.64, -53.66, 152.02, -3.675, -97.474, -0.262] to (266.79, -422.22, -4.17) mm, rotated rx 180 ry 0 rz 0 deg; joints [-3.642, -53.642, 152.048, -3.678, -97.519, -0.265]
  Set speed (50.8 mm/s)
  MoveL 732 to (267.42, -422.22, -4.17) mm, rotated rx 180 ry 0 rz 0 deg; joints [-3.645, -53.645, 152.092, -3.681, -97.561, -0.268]
  MoveC 733 to (267.87, -422.41, -4.18) mm, rotated rx 180 ry 0 rz 0 deg; joints [-3.659, -53.647, 152.122, -3.695, -97.589, -0.272] to (268.06, -422.86, -4.18) mm, rotated rx -180 ry 0 rz 0 deg; joints [-3.689, -53.647, 152.133, -3.726, -97.599, -0.277]
  MoveL 734 to (268.06, -448.26, -4.18) mm, rotated rx 180 ry 0 rz 0 deg; joints [-5.343, -53.628, 151.992, -5.392, -97.458, -0.511]
  MoveL 735 to (217.26, -448.26, -4.17) mm, rotated rx -180 ry 0 rz 0 deg; joints [-5.051, -53.245, 148.437, -5.069, -94.302, -0.186]
  MoveL 736 to (217.26, -397.46, -4.18) mm, rotated rx -180 ry 0 rz 0 deg; joints [-1.917, -53.295, 148.659, -1.927, -94.491, 0.092]
  MoveL 737 to (268.06, -397.46, -4.17) mm, rotated rx -180 ry 0 rz 0 deg; joints [-2.029, -53.664, 152.223, -2.051, -97.684, -0.033]
  MoveL 738 to (268.06, -422.86, -4.18) mm, rotated rx -180 ry 0 rz 0 deg; joints [-3.689, -53.647, 152.133, -3.726, -97.599, -0.277]
  MoveC 739 to (267.87, -423.31, -4.18) mm, rotated rx 180 ry 0 rz 0 deg; joints [-3.718, -53.646, 152.118, -3.754, -97.585, -0.28] to (267.42, -423.49, -4.18) mm, rotated rx 180 ry 0 rz 0 deg; joints [-3.728, -53.644, 152.086, -3.764, -97.555, -0.28]
  MoveL 740 to (266.79, -423.49, -4.18) mm, rotated rx -180 ry 0 rz 0 deg; joints [-3.725, -53.641, 152.042, -3.761, -97.514, -0.277]
  MoveC 741 to (266.34, -423.49, -3.99) mm, rotated rx -180 ry 0 rz 0 deg; joints [-3.723, -53.659, 152.014, -3.759, -97.468, -0.274] to (266.15, -423.49, -3.54) mm, rotated rx -180 ry 0 rz 0 deg; joints [-3.723, -53.707, 152.009, -3.758, -97.415, -0.27]
  Set speed (1000.0 mm/s)
  MoveL 742 to (266.15, -423.49, 5) mm, rotated rx 180 ry 0 rz 0 deg; joints [-3.725, -54.642, 152.161, -3.753, -96.633, -0.219]
  MoveL 743 to (266.15, -422.22, 5) mm, rotated rx 180 ry 0 rz 0 deg; joints [-3.642, -54.643, 152.167, -3.67, -96.639, -0.208]
  Set speed (25.4 mm/s)
  MoveL 744 to (266.15, -422.22, 1.83) mm, rotated rx 180 ry 0 rz 0 deg; joints [-3.641, -54.295, 152.111, -3.672, -96.931, -0.227]
  MoveL 745 to (266.15, -422.22, -7.72) mm, rotated rx -180 ry 0 rz 0 deg; joints [-3.639, -53.252, 151.938, -3.677, -97.799, -0.283]
  MoveC 746 to (266.34, -422.22, -8.16) mm, rotated rx -180 ry 0 rz 0 deg; joints [-3.639, -53.204, 151.942, -3.678, -97.851, -0.286] to (266.79, -422.22, -8.35) mm, rotated rx 180 ry 0 rz 0 deg; joints [-3.641, -53.185, 151.97, -3.68, -97.897, -0.289]
  Set speed (50.8 mm/s)
  MoveL 747 to (267.42, -422.22, -8.35) mm, rotated rx 180 ry 0 rz 0 deg; joints [-3.644, -53.188, 152.014, -3.683, -97.939, -0.292]
  MoveC 748 to (267.87, -422.41, -8.35) mm, rotated rx -180 ry 0 rz 0 deg; joints [-3.658, -53.189, 152.044, -3.697, -97.967, -0.296] to (268.06, -422.86, -8.35) mm, rotated rx -180 ry 0 rz 0 deg; joints [-3.688, -53.19, 152.055, -3.728, -97.977, -0.302]
  MoveL 749 to (268.06, -448.26, -8.35) mm, rotated rx 180 ry 0 rz 0 deg; joints [-5.342, -53.172, 151.914, -5.396, -97.835, -0.547]
  MoveL 750 to (217.26, -448.26, -8.35) mm, rotated rx -180 ry 0 rz 0 deg; joints [-5.05, -52.823, 148.365, -5.07, -94.651, -0.217]
  MoveL 751 to (217.26, -397.46, -8.35) mm, rotated rx -180 ry 0 rz 0 deg; joints [-1.916, -52.872, 148.587, -1.927, -94.842, 0.08]
  MoveL 752 to (268.06, -397.46, -8.35) mm, rotated rx -180 ry 0 rz 0 deg; joints [-2.028, -53.206, 152.145, -2.052, -98.064, -0.047]
  MoveL 753 to (268.06, -422.86, -8.35) mm, rotated rx -180 ry 0 rz 0 deg; joints [-3.688, -53.19, 152.055, -3.728, -97.977, -0.302]
  MoveC 754 to (267.87, -423.31, -8.35) mm, rotated rx -180 ry 0 rz 0 deg; joints [-3.717, -53.189, 152.04, -3.756, -97.963, -0.305] to (267.42, -423.49, -8.35) mm, rotated rx -180 ry 0 rz 0 deg; joints [-3.727, -53.187, 152.008, -3.767, -97.933, -0.305]
  MoveL 755 to (266.79, -423.49, -8.35) mm, rotated rx 180 ry 0 rz 0 deg; joints [-3.724, -53.184, 151.964, -3.763, -97.892, -0.302]
  MoveC 756 to (266.34, -423.49, -8.16) mm, rotated rx 180 ry 0 rz 0 deg; joints [-3.722, -53.203, 151.936, -3.761, -97.846, -0.298] to (266.15, -423.49, -7.72) mm, rotated rx -180 ry 0 rz 0 deg; joints [-3.722, -53.251, 151.932, -3.76, -97.793, -0.295]
  Set speed (1000.0 mm/s)
  MoveL 757 to (266.15, -423.49, 6) mm, rotated rx -180 ry 0 rz 0 deg; joints [-3.725, -54.752, 152.178, -3.753, -96.541, -0.212]
  MoveL 758 to (139.15, -422.22, 6) mm, rotated rx -180 ry 0 rz 0 deg; joints [-3.182, -53.164, 143.134, -3.186, -89.101, 0.274]
  Set speed (25.4 mm/s)
  MoveL 759 to (139.15, -422.22, -3.54) mm, rotated rx -180 ry 0 rz 0 deg; joints [-3.18, -52.299, 142.992, -3.183, -89.823, 0.234]
  MoveC 760 to (139.34, -422.22, -3.99) mm, rotated rx -180 ry 0 rz 0 deg; joints [-3.18, -52.261, 142.999, -3.184, -89.867, 0.231] to (139.79, -422.22, -4.17) mm, rotated rx 180 ry 0 rz 0 deg; joints [-3.182, -52.252, 143.028, -3.185, -89.906, 0.229]
  Set speed (50.8 mm/s)
  MoveL 761 to (140.42, -422.22, -4.17) mm, rotated rx -180 ry 0 rz 0 deg; joints [-3.184, -52.262, 143.074, -3.187, -89.942, 0.227]
  MoveC 762 to (140.87, -422.41, -4.17) mm, rotated rx 180 ry 0 rz 0 deg; joints [-3.196, -52.269, 143.106, -3.199, -89.966, 0.226] to (141.06, -422.86, -4.17) mm, rotated rx 180 ry 0 rz 0 deg; joints [-3.222, -52.271, 143.118, -3.226, -89.976, 0.225]
  MoveL 763 to (141.06, -448.26, -4.18) mm, rotated rx 180 ry 0 rz 0 deg; joints [-4.668, -52.234, 142.989, -4.672, -89.883, 0.211]
  MoveL 764 to (90.26, -448.26, -4.18) mm, rotated rx -180 ry 0 rz 0 deg; joints [-4.443, -51.328, 139.277, -4.453, -87.086, 0.432]
  MoveL 765 to (90.26, -397.46, -4.18) mm, rotated rx -180 ry 0 rz 0 deg; joints [-1.686, -51.397, 139.481, -1.692, -87.215, 0.329]
  MoveL 766 to (141.06, -397.46, -4.18) mm, rotated rx -180 ry 0 rz 0 deg; joints [-1.771, -52.299, 143.2, -1.775, -90.031, 0.244]
  MoveL 767 to (141.06, -422.86, -4.17) mm, rotated rx 180 ry 0 rz 0 deg; joints [-3.222, -52.271, 143.118, -3.226, -89.976, 0.225]
  MoveC 768 to (140.87, -423.31, -4.18) mm, rotated rx 180 ry 0 rz 0 deg; joints [-3.247, -52.268, 143.102, -3.251, -89.964, 0.225] to (140.42, -423.49, -4.17) mm, rotated rx -180 ry 0 rz 0 deg; joints [-3.256, -52.26, 143.069, -3.26, -89.938, 0.226]
  MoveL 769 to (139.79, -423.49, -4.18) mm, rotated rx 180 ry 0 rz 0 deg; joints [-3.254, -52.25, 143.023, -3.258, -89.902, 0.228]
  MoveC 770 to (139.34, -423.49, -3.99) mm, rotated rx -180 ry 0 rz 0 deg; joints [-3.252, -52.26, 142.993, -3.256, -89.863, 0.231] to (139.15, -423.49, -3.54) mm, rotated rx 180 ry 0 rz 0 deg; joints [-3.252, -52.297, 142.987, -3.256, -89.819, 0.233]
  Set speed (1000.0 mm/s)
  MoveL 771 to (139.15, -423.49, 5) mm, rotated rx -180 ry 0 rz 0 deg; joints [-3.254, -53.071, 143.114, -3.258, -89.173, 0.27]
  MoveL 772 to (139.15, -422.22, 5) mm, rotated rx -180 ry 0 rz 0 deg; joints [-3.182, -53.073, 143.119, -3.186, -89.177, 0.27]
  Set speed (25.4 mm/s)
  MoveL 773 to (139.15, -422.22, 1.83) mm, rotated rx -180 ry 0 rz 0 deg; joints [-3.181, -52.785, 143.073, -3.185, -89.418, 0.256]
  MoveL 774 to (139.15, -422.22, -7.72) mm, rotated rx -180 ry 0 rz 0 deg; joints [-3.179, -51.92, 142.927, -3.183, -90.135, 0.216]
  MoveC 775 to (139.34, -422.22, -8.16) mm, rotated rx 180 ry 0 rz 0 deg; joints [-3.179, -51.883, 142.933, -3.183, -90.179, 0.214] to (139.79, -422.22, -8.35) mm, rotated rx -180 ry 0 rz 0 deg; joints [-3.181, -51.873, 142.963, -3.184, -90.219, 0.212]
  Set speed (50.8 mm/s)
  MoveL 776 to (140.42, -422.22, -8.35) mm, rotated rx -180 ry 0 rz 0 deg; joints [-3.183, -51.883, 143.009, -3.186, -90.255, 0.21]
  MoveC 777 to (140.87, -422.41, -8.35) mm, rotated rx 180 ry 0 rz 0 deg; joints [-3.195, -51.89, 143.041, -3.198, -90.28, 0.208] to (141.06, -422.86, -8.35) mm, rotated rx -180 ry 0 rz 0 deg; joints [-3.221, -51.892, 143.052, -3.225, -90.289, 0.207]
  MoveL 778 to (141.06, -448.26, -8.35) mm, rotated rx -180 ry 0 rz 0 deg; joints [-4.667, -51.856, 142.924, -4.671, -90.195, 0.185]
  MoveL 779 to (90.26, -448.26, -8.35) mm, rotated rx -180 ry 0 rz 0 deg; joints [-4.443, -50.973, 139.215, -4.451, -87.377, 0.409]
  MoveL 780 to (90.26, -397.46, -8.35) mm, rotated rx -180 ry 0 rz 0 deg; joints [-1.685, -51.042, 139.419, -1.69, -87.508, 0.32]
  MoveL 781 to (141.06, -397.46, -8.35) mm, rotated rx -180 ry 0 rz 0 deg; joints [-1.77, -51.919, 143.134, -1.774, -90.346, 0.235]
  MoveL 782 to (141.06, -422.86, -8.35) mm, rotated rx -180 ry 0 rz 0 deg; joints [-3.221, -51.892, 143.052, -3.225, -90.289, 0.207]
  MoveC 783 to (140.87, -423.31, -8.35) mm, rotated rx -180 ry 0 rz 0 deg; joints [-3.246, -51.888, 143.037, -3.25, -90.277, 0.207] to (140.42, -423.49, -8.35) mm, rotated rx -180 ry 0 rz 0 deg; joints [-3.255, -51.881, 143.004, -3.259, -90.251, 0.209]
  MoveL 784 to (139.79, -423.49, -8.35) mm, rotated rx -180 ry 0 rz 0 deg; joints [-3.253, -51.871, 142.958, -3.257, -90.215, 0.211]
  MoveC 785 to (139.34, -423.49, -8.16) mm, rotated rx 180 ry 0 rz 0 deg; joints [-3.252, -51.881, 142.928, -3.255, -90.176, 0.213] to (139.15, -423.49, -7.72) mm, rotated rx 180 ry 0 rz 0 deg; joints [-3.251, -51.919, 142.922, -3.255, -90.132, 0.215]
  Set speed (1000.0 mm/s)
  MoveL 786 to (139.15, -423.49, 6) mm, rotated rx 180 ry 0 rz 0 deg; joints [-3.254, -53.162, 143.129, -3.258, -89.097, 0.274]
  MoveL 787 to (-92.16, -422.22, 6) mm, rotated rx 180 ry 0 rz 0 deg; joints [-2.586, -47.662, 125.571, -2.657, -77.052, 0.829]
  Set speed (25.4 mm/s)
  MoveL 788 to (-92.16, -422.22, -3.54) mm, rotated rx -180 ry 0 rz 0 deg; joints [-2.584, -47.005, 125.456, -2.65, -77.594, 0.803]
  MoveC 789 to (-91.98, -422.22, -3.99) mm, rotated rx -180 ry 0 rz 0 deg; joints [-2.584, -46.979, 125.465, -2.65, -77.629, 0.801] to (-91.53, -422.22, -4.17) mm, rotated rx -180 ry 0 rz 0 deg; joints [-2.585, -46.979, 125.499, -2.65, -77.662, 0.8]
  Set speed (50.8 mm/s)
  MoveL 790 to (-90.89, -422.22, -4.18) mm, rotated rx 180 ry 0 rz 0 deg; joints [-2.587, -46.997, 125.549, -2.651, -77.695, 0.798]
  MoveC 791 to (-90.44, -422.41, -4.18) mm, rotated rx 180 ry 0 rz 0 deg; joints [-2.596, -47.009, 125.584, -2.661, -77.717, 0.799] to (-90.26, -422.86, -4.17) mm, rotated rx -180 ry 0 rz 0 deg; joints [-2.617, -47.014, 125.597, -2.683, -77.726, 0.803]
  MoveL 792 to (-90.26, -448.26, -4.17) mm, rotated rx -180 ry 0 rz 0 deg; joints [-3.794, -46.967, 125.483, -3.888, -77.672, 1.046]
  MoveL 793 to (-141.06, -448.26, -4.18) mm, rotated rx -180 ry 0 rz 0 deg; joints [-3.644, -45.471, 121.399, -3.775, -75.088, 1.19]
  MoveL 794 to (-141.06, -397.46, -4.17) mm, rotated rx -180 ry 0 rz 0 deg; joints [-1.381, -45.553, 121.584, -1.433, -75.165, 0.618]
  MoveL 795 to (-90.26, -397.46, -4.17) mm, rotated rx -180 ry 0 rz 0 deg; joints [-1.438, -47.047, 125.67, -1.476, -77.757, 0.563]
  MoveL 796 to (-90.26, -422.86, -4.17) mm, rotated rx -180 ry 0 rz 0 deg; joints [-2.617, -47.014, 125.597, -2.683, -77.726, 0.803]
  MoveC 797 to (-90.44, -423.31, -4.18) mm, rotated rx 180 ry 0 rz 0 deg; joints [-2.638, -47.008, 125.581, -2.704, -77.716, 0.808] to (-90.89, -423.49, -4.18) mm, rotated rx -180 ry 0 rz 0 deg; joints [-2.646, -46.995, 125.544, -2.712, -77.692, 0.811]
  MoveL 798 to (-91.53, -423.49, -4.18) mm, rotated rx 180 ry 0 rz 0 deg; joints [-2.644, -46.977, 125.494, -2.711, -77.66, 0.812]
  MoveC 799 to (-91.98, -423.49, -3.99) mm, rotated rx -180 ry 0 rz 0 deg; joints [-2.643, -46.977, 125.46, -2.71, -77.627, 0.813] to (-92.16, -423.49, -3.54) mm, rotated rx -180 ry 0 rz 0 deg; joints [-2.643, -47.003, 125.451, -2.71, -77.592, 0.815]
  Set speed (1000.0 mm/s)
  MoveL 800 to (-92.16, -423.49, 5) mm, rotated rx -180 ry 0 rz 0 deg; joints [-2.645, -47.591, 125.555, -2.717, -77.107, 0.839]
  MoveL 801 to (-92.16, -422.22, 5) mm, rotated rx -180 ry 0 rz 0 deg; joints [-2.586, -47.593, 125.559, -2.657, -77.109, 0.826]
  Set speed (25.4 mm/s)
  MoveL 802 to (-92.16, -422.22, 1.83) mm, rotated rx 180 ry 0 rz 0 deg; joints [-2.585, -47.374, 125.522, -2.654, -77.29, 0.817]
  MoveL 803 to (-92.16, -422.22, -7.71) mm, rotated rx -180 ry 0 rz 0 deg; joints [-2.583, -46.716, 125.403, -2.647, -77.829, 0.791]
  MoveC 804 to (-91.98, -422.22, -8.16) mm, rotated rx -180 ry 0 rz 0 deg; joints [-2.584, -46.691, 125.412, -2.647, -77.864, 0.79] to (-91.53, -422.22, -8.35) mm, rotated rx 180 ry 0 rz 0 deg; joints [-2.585, -46.69, 125.445, -2.647, -77.897, 0.788]
  Set speed (50.8 mm/s)
  MoveL 805 to (-90.89, -422.22, -8.35) mm, rotated rx -180 ry 0 rz 0 deg; joints [-2.586, -46.708, 125.496, -2.648, -77.93, 0.787]
  MoveC 806 to (-90.44, -422.41, -8.35) mm, rotated rx -180 ry 0 rz 0 deg; joints [-2.595, -46.721, 125.531, -2.658, -77.953, 0.788] to (-90.26, -422.86, -8.35) mm, rotated rx -180 ry 0 rz 0 deg; joints [-2.617, -46.725, 125.544, -2.679, -77.961, 0.792]
  MoveL 807 to (-90.26, -448.26, -8.35) mm, rotated rx -180 ry 0 rz 0 deg; joints [-3.794, -46.678, 125.43, -3.884, -77.907, 1.029]
  MoveL 808 to (-141.06, -448.26, -8.35) mm, rotated rx -180 ry 0 rz 0 deg; joints [-3.644, -45.197, 121.348, -3.771, -75.31, 1.174]
  MoveL 809 to (-141.06, -397.46, -8.35) mm, rotated rx -180 ry 0 rz 0 deg; joints [-1.381, -45.278, 121.532, -1.431, -75.389, 0.612]
  MoveL 810 to (-90.26, -397.46, -8.35) mm, rotated rx 180 ry 0 rz 0 deg; joints [-1.438, -46.758, 125.617, -1.474, -77.993, 0.557]
  MoveL 811 to (-90.26, -422.86, -8.35) mm, rotated rx -180 ry 0 rz 0 deg; joints [-2.617, -46.725, 125.544, -2.679, -77.961, 0.792]
  MoveC 812 to (-90.44, -423.31, -8.35) mm, rotated rx 180 ry 0 rz 0 deg; joints [-2.637, -46.719, 125.528, -2.7, -77.951, 0.796] to (-90.89, -423.49, -8.35) mm, rotated rx 180 ry 0 rz 0 deg; joints [-2.645, -46.706, 125.491, -2.709, -77.928, 0.799]
  MoveL 813 to (-91.53, -423.49, -8.35) mm, rotated rx -180 ry 0 rz 0 deg; joints [-2.643, -46.688, 125.441, -2.707, -77.895, 0.8]
  MoveC 814 to (-91.98, -423.49, -8.16) mm, rotated rx 180 ry 0 rz 0 deg; joints [-2.642, -46.689, 125.408, -2.707, -77.862, 0.802] to (-92.16, -423.49, -7.72) mm, rotated rx -180 ry 0 rz 0 deg; joints [-2.642, -46.714, 125.399, -2.707, -77.827, 0.803]
  Set speed (1000.0 mm/s)
  MoveL 815 to (-92.16, -423.49, 6) mm, rotated rx -180 ry 0 rz 0 deg; joints [-2.645, -47.66, 125.566, -2.718, -77.05, 0.842]
  MoveL 816 to (-219.16, -422.22, 6) mm, rotated rx -180 ry 0 rz 0 deg; joints [-2.345, -43.635, 115.134, -2.489, -70.646, 1.062]
  Set speed (25.4 mm/s)
  MoveL 817 to (-219.16, -422.22, -3.54) mm, rotated rx -180 ry 0 rz 0 deg; joints [-2.343, -43.053, 115.027, -2.48, -71.12, 1.04]
  MoveC 818 to (-218.98, -422.22, -3.99) mm, rotated rx -180 ry 0 rz 0 deg; joints [-2.343, -43.032, 115.038, -2.48, -71.152, 1.038] to (-218.53, -422.22, -4.17) mm, rotated rx -180 ry 0 rz 0 deg; joints [-2.344, -43.036, 115.074, -2.481, -71.184, 1.037]
  Set speed (50.8 mm/s)
  MoveL 819 to (-217.89, -422.22, -4.17) mm, rotated rx 180 ry 0 rz 0 deg; joints [-2.345, -43.057, 115.128, -2.481, -71.216, 1.036]
  MoveC 820 to (-217.44, -422.41, -4.17) mm, rotated rx -180 ry 0 rz 0 deg; joints [-2.354, -43.072, 115.165, -2.49, -71.239, 1.038] to (-217.26, -422.86, -4.18) mm, rotated rx 180 ry 0 rz 0 deg; joints [-2.373, -43.078, 115.179, -2.51, -71.248, 1.044]
  MoveL 821 to (-217.26, -448.26, -4.18) mm, rotated rx 180 ry 0 rz 0 deg; joints [-3.44, -43.028, 115.068, -3.638, -71.205, 1.394]
  MoveL 822 to (-268.06, -448.26, -4.17) mm, rotated rx -180 ry 0 rz 0 deg; joints [-3.317, -41.266, 110.69, -3.567, -68.59, 1.525]
  MoveL 823 to (-268.06, -397.46, -4.18) mm, rotated rx -180 ry 0 rz 0 deg; joints [-1.257, -41.351, 110.87, -1.353, -68.655, 0.746]
  MoveL 824 to (-217.26, -397.46, -4.17) mm, rotated rx 180 ry 0 rz 0 deg; joints [-1.304, -43.112, 115.25, -1.381, -71.273, 0.696]
  MoveL 825 to (-217.26, -422.86, -4.18) mm, rotated rx 180 ry 0 rz 0 deg; joints [-2.373, -43.078, 115.179, -2.51, -71.248, 1.044]
  MoveC 826 to (-217.44, -423.31, -4.17) mm, rotated rx 180 ry 0 rz 0 deg; joints [-2.391, -43.071, 115.162, -2.53, -71.238, 1.05] to (-217.89, -423.49, -4.17) mm, rotated rx -180 ry 0 rz 0 deg; joints [-2.399, -43.055, 115.123, -2.538, -71.215, 1.054]
  MoveL 827 to (-218.53, -423.49, -4.17) mm, rotated rx -180 ry 0 rz 0 deg; joints [-2.397, -43.034, 115.069, -2.537, -71.182, 1.055]
  MoveC 828 to (-218.98, -423.49, -3.99) mm, rotated rx 180 ry 0 rz 0 deg; joints [-2.397, -43.03, 115.033, -2.537, -71.15, 1.056] to (-219.16, -423.49, -3.54) mm, rotated rx 180 ry 0 rz 0 deg; joints [-2.396, -43.051, 115.023, -2.537, -71.118, 1.057]
  Set speed (1000.0 mm/s)
  MoveL 829 to (-219.16, -423.49, 5) mm, rotated rx 180 ry 0 rz 0 deg; joints [-2.398, -43.572, 115.119, -2.545, -70.695, 1.078]
  MoveL 830 to (-219.16, -422.22, 5) mm, rotated rx 180 ry 0 rz 0 deg; joints [-2.345, -43.574, 115.124, -2.488, -70.696, 1.06]
  Set speed (25.4 mm/s)
  MoveL 831 to (-219.16, -422.22, 1.82) mm, rotated rx -180 ry 0 rz 0 deg; joints [-2.344, -43.381, 115.088, -2.485, -70.854, 1.052]
  MoveL 832 to (-219.16, -422.22, -7.72) mm, rotated rx -180 ry 0 rz 0 deg; joints [-2.342, -42.798, 114.978, -2.477, -71.326, 1.03]
  MoveC 833 to (-218.98, -422.22, -8.16) mm, rotated rx 180 ry 0 rz 0 deg; joints [-2.343, -42.777, 114.988, -2.476, -71.357, 1.029] to (-218.53, -422.22, -8.35) mm, rotated rx -180 ry 0 rz 0 deg; joints [-2.343, -42.781, 115.024, -2.477, -71.389, 1.028]
  Set speed (50.8 mm/s)
  MoveL 834 to (-217.89, -422.22, -8.35) mm, rotated rx -180 ry 0 rz 0 deg; joints [-2.344, -42.802, 115.078, -2.477, -71.422, 1.026]
  MoveC 835 to (-217.44, -422.41, -8.35) mm, rotated rx -180 ry 0 rz 0 deg; joints [-2.353, -42.816, 115.115, -2.486, -71.445, 1.028] to (-217.26, -422.86, -8.35) mm, rotated rx -180 ry 0 rz 0 deg; joints [-2.372, -42.822, 115.13, -2.506, -71.454, 1.034]
  MoveL 836 to (-217.26, -448.26, -8.35) mm, rotated rx -180 ry 0 rz 0 deg; joints [-3.44, -42.773, 115.019, -3.633, -71.41, 1.38]
  MoveL 837 to (-268.06, -448.26, -8.35) mm, rotated rx -180 ry 0 rz 0 deg; joints [-3.316, -41.022, 110.641, -3.561, -68.786, 1.512]
  MoveL 838 to (-268.06, -397.46, -8.35) mm, rotated rx 180 ry 0 rz 0 deg; joints [-1.256, -41.106, 110.821, -1.351, -68.851, 0.741]
  MoveL 839 to (-217.26, -397.46, -8.35) mm, rotated rx -180 ry 0 rz 0 deg; joints [-1.303, -42.856, 115.2, -1.378, -71.48, 0.69]
  MoveL 840 to (-217.26, -422.86, -8.35) mm, rotated rx -180 ry 0 rz 0 deg; joints [-2.372, -42.822, 115.13, -2.506, -71.454, 1.034]
  MoveC 841 to (-217.44, -423.31, -8.35) mm, rotated rx -180 ry 0 rz 0 deg; joints [-2.391, -42.815, 115.112, -2.526, -71.444, 1.04] to (-217.89, -423.49, -8.35) mm, rotated rx -180 ry 0 rz 0 deg; joints [-2.398, -42.8, 115.073, -2.534, -71.42, 1.044]
  MoveL 842 to (-218.53, -423.49, -8.35) mm, rotated rx -180 ry 0 rz 0 deg; joints [-2.397, -42.778, 115.02, -2.533, -71.388, 1.045]
  MoveC 843 to (-218.98, -423.49, -8.16) mm, rotated rx -180 ry 0 rz 0 deg; joints [-2.396, -42.775, 114.984, -2.533, -71.355, 1.046] to (-219.16, -423.49, -7.72) mm, rotated rx 180 ry 0 rz 0 deg; joints [-2.396, -42.796, 114.973, -2.533, -71.324, 1.047]
  Set speed (1000.0 mm/s)
  MoveL 844 to (-219.16, -423.49, 6) mm, rotated rx 180 ry 0 rz 0 deg; joints [-2.398, -43.633, 115.13, -2.546, -70.645, 1.08]
  MoveL 845 to (-346.16, -422.22, 6) mm, rotated rx 180 ry 0 rz 0 deg; joints [-2.145, -38.951, 103.885, -2.389, -64.084, 1.284]
  Set speed (25.4 mm/s)
  MoveL 846 to (-346.16, -422.22, -3.54) mm, rotated rx -180 ry 0 rz 0 deg; joints [-2.143, -38.428, 103.781, -2.379, -64.502, 1.264]
  MoveC 847 to (-345.98, -422.22, -3.99) mm, rotated rx 180 ry 0 rz 0 deg; joints [-2.143, -38.41, 103.793, -2.378, -64.532, 1.263] to (-345.53, -422.22, -4.17) mm, rotated rx 180 ry 0 rz 0 deg; joints [-2.144, -38.418, 103.833, -2.378, -64.564, 1.262]
  Set speed (50.8 mm/s)
  MoveL 848 to (-344.89, -422.22, -4.18) mm, rotated rx -180 ry 0 rz 0 deg; joints [-2.145, -38.443, 103.891, -2.379, -64.598, 1.261]
  MoveC 849 to (-344.44, -422.41, -4.17) mm, rotated rx -180 ry 0 rz 0 deg; joints [-2.153, -38.46, 103.932, -2.387, -64.621, 1.263] to (-344.26, -422.86, -4.18) mm, rotated rx -180 ry 0 rz 0 deg; joints [-2.17, -38.466, 103.948, -2.406, -64.631, 1.271]
  MoveL 850 to (-344.26, -448.26, -4.17) mm, rotated rx 180 ry 0 rz 0 deg; joints [-3.147, -38.414, 103.837, -3.488, -64.593, 1.723]
  MoveL 851 to (-395.06, -448.26, -4.17) mm, rotated rx 180 ry 0 rz 0 deg; joints [-3.043, -36.363, 99.045, -3.456, -61.854, 1.858]
  MoveL 852 to (-395.06, -397.46, -4.18) mm, rotated rx -180 ry 0 rz 0 deg; joints [-1.153, -36.452, 99.227, -1.311, -61.911, 0.872]
  MoveL 853 to (-344.26, -397.46, -4.18) mm, rotated rx -180 ry 0 rz 0 deg; joints [-1.192, -38.502, 104.018, -1.323, -64.653, 0.821]
  MoveL 854 to (-344.26, -422.86, -4.18) mm, rotated rx -180 ry 0 rz 0 deg; joints [-2.17, -38.466, 103.948, -2.406, -64.631, 1.271]
  MoveC 855 to (-344.44, -423.31, -4.17) mm, rotated rx 180 ry 0 rz 0 deg; joints [-2.187, -38.458, 103.929, -2.425, -64.62, 1.279] to (-344.89, -423.49, -4.18) mm, rotated rx -180 ry 0 rz 0 deg; joints [-2.194, -38.44, 103.887, -2.433, -64.596, 1.283]
  MoveL 856 to (-345.53, -423.49, -4.18) mm, rotated rx -180 ry 0 rz 0 deg; joints [-2.193, -38.416, 103.828, -2.432, -64.562, 1.284]
  MoveC 857 to (-345.98, -423.49, -3.99) mm, rotated rx -180 ry 0 rz 0 deg; joints [-2.192, -38.408, 103.789, -2.432, -64.53, 1.286] to (-346.16, -423.49, -3.54) mm, rotated rx -180 ry 0 rz 0 deg; joints [-2.192, -38.426, 103.776, -2.433, -64.501, 1.287]
  Set speed (1000.0 mm/s)
  MoveL 858 to (-346.16, -423.49, 5) mm, rotated rx -180 ry 0 rz 0 deg; joints [-2.193, -38.894, 103.87, -2.442, -64.126, 1.305]
  MoveL 859 to (-346.16, -422.22, 5) mm, rotated rx 180 ry 0 rz 0 deg; joints [-2.144, -38.896, 103.874, -2.388, -64.128, 1.282]
  Set speed (25.4 mm/s)
  MoveL 860 to (-346.16, -422.22, 1.82) mm, rotated rx 180 ry 0 rz 0 deg; joints [-2.144, -38.722, 103.84, -2.384, -64.267, 1.275]
  MoveL 861 to (-346.16, -422.22, -7.71) mm, rotated rx -180 ry 0 rz 0 deg; joints [-2.142, -38.198, 103.733, -2.374, -64.684, 1.256]
  MoveC 862 to (-345.98, -422.22, -8.16) mm, rotated rx -180 ry 0 rz 0 deg; joints [-2.143, -38.181, 103.745, -2.374, -64.714, 1.254] to (-345.53, -422.22, -8.35) mm, rotated rx -180 ry 0 rz 0 deg; joints [-2.143, -38.188, 103.785, -2.374, -64.746, 1.253]
  Set speed (50.8 mm/s)
  MoveL 863 to (-344.89, -422.22, -8.35) mm, rotated rx -180 ry 0 rz 0 deg; joints [-2.144, -38.213, 103.843, -2.374, -64.78, 1.252]
  MoveC 864 to (-344.44, -422.41, -8.35) mm, rotated rx -180 ry 0 rz 0 deg; joints [-2.152, -38.23, 103.884, -2.383, -64.803, 1.254] to (-344.26, -422.86, -8.35) mm, rotated rx 180 ry 0 rz 0 deg; joints [-2.169, -38.236, 103.9, -2.402, -64.813, 1.262]
  MoveL 865 to (-344.26, -448.26, -8.35) mm, rotated rx -180 ry 0 rz 0 deg; joints [-3.146, -38.185, 103.789, -3.482, -64.775, 1.71]
  MoveL 866 to (-395.06, -448.26, -8.35) mm, rotated rx -180 ry 0 rz 0 deg; joints [-3.042, -36.142, 98.997, -3.45, -62.027, 1.846]
  MoveL 867 to (-395.06, -397.46, -8.35) mm, rotated rx -180 ry 0 rz 0 deg; joints [-1.152, -36.231, 99.179, -1.308, -62.085, 0.867]
  MoveL 868 to (-344.26, -397.46, -8.35) mm, rotated rx 180 ry 0 rz 0 deg; joints [-1.191, -38.271, 103.97, -1.321, -64.835, 0.816]
  MoveL 869 to (-344.26, -422.86, -8.35) mm, rotated rx 180 ry 0 rz 0 deg; joints [-2.169, -38.236, 103.9, -2.402, -64.813, 1.262]
  MoveC 870 to (-344.44, -423.31, -8.35) mm, rotated rx -180 ry 0 rz 0 deg; joints [-2.186, -38.228, 103.881, -2.421, -64.802, 1.27] to (-344.89, -423.49, -8.35) mm, rotated rx -180 ry 0 rz 0 deg; joints [-2.193, -38.21, 103.839, -2.428, -64.778, 1.274]
  MoveL 871 to (-345.53, -423.49, -8.35) mm, rotated rx 180 ry 0 rz 0 deg; joints [-2.192, -38.186, 103.78, -2.428, -64.744, 1.275]
  MoveC 872 to (-345.98, -423.49, -8.16) mm, rotated rx -180 ry 0 rz 0 deg; joints [-2.191, -38.178, 103.741, -2.428, -64.712, 1.277] to (-346.16, -423.49, -7.72) mm, rotated rx -180 ry 0 rz 0 deg; joints [-2.191, -38.196, 103.729, -2.428, -64.683, 1.278]
  Set speed (1000.0 mm/s)
  MoveL 873 to (-346.16, -423.49, 6) mm, rotated rx 180 ry 0 rz 0 deg; joints [-2.193, -38.948, 103.88, -2.443, -64.082, 1.307]
  MoveL 874 to (-346.16, -235.89, 6) mm, rotated rx 180 ry 0 rz 0 deg; joints [5.013, -38.817, 103.463, 5.58, -63.88, -2.114]
  Set speed (25.4 mm/s)
  MoveL 875 to (-346.16, -235.88, -3.54) mm, rotated rx -180 ry 0 rz 0 deg; joints [5.015, -38.296, 103.359, 5.562, -64.295, -2.07]
  MoveC 876 to (-345.98, -235.89, -3.99) mm, rotated rx -180 ry 0 rz 0 deg; joints [5.016, -38.279, 103.371, 5.562, -64.325, -2.067] to (-345.53, -235.89, -4.17) mm, rotated rx 180 ry 0 rz 0 deg; joints [5.018, -38.287, 103.41, 5.562, -64.357, -2.065]
  Set speed (50.8 mm/s)
  MoveL 877 to (-344.89, -235.88, -4.18) mm, rotated rx -180 ry 0 rz 0 deg; joints [5.02, -38.312, 103.469, 5.563, -64.39, -2.062]
  MoveC 878 to (-344.44, -236.07, -4.17) mm, rotated rx 180 ry 0 rz 0 deg; joints [5.014, -38.33, 103.512, 5.556, -64.415, -2.057] to (-344.26, -236.52, -4.18) mm, rotated rx -180 ry 0 rz 0 deg; joints [4.998, -38.338, 103.533, 5.537, -64.426, -2.048]
  MoveL 879 to (-344.26, -261.92, -4.17) mm, rotated rx 180 ry 0 rz 0 deg; joints [4.025, -38.409, 103.716, 4.455, -64.503, -1.587]
  MoveL 880 to (-395.06, -261.92, -4.18) mm, rotated rx -180 ry 0 rz 0 deg; joints [3.892, -36.354, 98.923, 4.414, -61.768, -1.76]
  MoveL 881 to (-395.06, -211.12, -4.18) mm, rotated rx -180 ry 0 rz 0 deg; joints [5.772, -36.191, 98.512, 6.559, -61.605, -2.77]
  MoveL 882 to (-344.26, -211.12, -4.18) mm, rotated rx 180 ry 0 rz 0 deg; joints [5.967, -38.251, 103.31, 6.618, -64.334, -2.514]
  MoveL 883 to (-344.26, -236.52, -4.18) mm, rotated rx -180 ry 0 rz 0 deg; joints [4.998, -38.338, 103.533, 5.537, -64.426, -2.048]
  MoveC 884 to (-344.44, -236.97, -4.18) mm, rotated rx -180 ry 0 rz 0 deg; joints [4.98, -38.333, 103.519, 5.517, -64.418, -2.04] to (-344.89, -237.16, -4.18) mm, rotated rx -180 ry 0 rz 0 deg; joints [4.971, -38.315, 103.479, 5.509, -64.395, -2.039]
  MoveL 885 to (-345.53, -237.16, -4.18) mm, rotated rx 180 ry 0 rz 0 deg; joints [4.969, -38.291, 103.421, 5.508, -64.361, -2.041]
  MoveC 886 to (-345.98, -237.16, -3.99) mm, rotated rx -180 ry 0 rz 0 deg; joints [4.967, -38.283, 103.381, 5.508, -64.329, -2.044] to (-346.16, -237.16, -3.54) mm, rotated rx -180 ry 0 rz 0 deg; joints [4.967, -38.3, 103.369, 5.508, -64.3, -2.047]
  Set speed (1000.0 mm/s)
  MoveL 887 to (-346.16, -237.16, 5) mm, rotated rx -180 ry 0 rz 0 deg; joints [4.965, -38.767, 103.462, 5.524, -63.928, -2.086]
  MoveL 888 to (-346.16, -235.89, 5) mm, rotated rx 180 ry 0 rz 0 deg; joints [5.013, -38.763, 103.452, 5.578, -63.924, -2.11]
  Set speed (25.4 mm/s)
  MoveL 889 to (-346.16, -235.89, 1.83) mm, rotated rx 180 ry 0 rz 0 deg; joints [5.014, -38.59, 103.418, 5.572, -64.062, -2.095]
  MoveL 890 to (-346.16, -235.88, -7.72) mm, rotated rx -180 ry 0 rz 0 deg; joints [5.016, -38.068, 103.311, 5.555, -64.476, -2.051]
  MoveC 891 to (-345.98, -235.88, -8.16) mm, rotated rx -180 ry 0 rz 0 deg; joints [5.017, -38.05, 103.323, 5.555, -64.505, -2.048] to (-345.53, -235.89, -8.35) mm, rotated rx -180 ry 0 rz 0 deg; joints [5.018, -38.058, 103.363, 5.555, -64.537, -2.046]
  Set speed (50.8 mm/s)
  MoveL 892 to (-344.89, -235.88, -8.35) mm, rotated rx -180 ry 0 rz 0 deg; joints [5.021, -38.082, 103.421, 5.556, -64.571, -2.043]
  MoveC 893 to (-344.44, -236.07, -8.35) mm, rotated rx 180 ry 0 rz 0 deg; joints [5.015, -38.101, 103.464, 5.548, -64.595, -2.038] to (-344.26, -236.52, -8.35) mm, rotated rx -180 ry 0 rz 0 deg; joints [4.998, -38.109, 103.485, 5.529, -64.607, -2.029]
  MoveL 894 to (-344.26, -261.92, -8.35) mm, rotated rx -180 ry 0 rz 0 deg; joints [4.026, -38.179, 103.669, 4.449, -64.685, -1.572]
  MoveL 895 to (-395.06, -261.92, -8.35) mm, rotated rx -180 ry 0 rz 0 deg; joints [3.893, -36.133, 98.875, 4.407, -61.941, -1.745]
  MoveL 896 to (-395.06, -211.12, -8.35) mm, rotated rx 180 ry 0 rz 0 deg; joints [5.773, -35.971, 98.464, 6.549, -61.776, -2.748]
  MoveL 897 to (-344.26, -211.12, -8.35) mm, rotated rx -180 ry 0 rz 0 deg; joints [5.968, -38.023, 103.262, 6.609, -64.514, -2.491]
  MoveL 898 to (-344.26, -236.52, -8.35) mm, rotated rx -180 ry 0 rz 0 deg; joints [4.998, -38.109, 103.485, 5.529, -64.607, -2.029]
  MoveC 899 to (-344.44, -236.97, -8.35) mm, rotated rx 180 ry 0 rz 0 deg; joints [4.981, -38.103, 103.472, 5.51, -64.598, -2.022] to (-344.89, -237.16, -8.35) mm, rotated rx -180 ry 0 rz 0 deg; joints [4.972, -38.086, 103.431, 5.502, -64.575, -2.02]
  MoveL 900 to (-345.53, -237.16, -8.35) mm, rotated rx -180 ry 0 rz 0 deg; joints [4.97, -38.061, 103.373, 5.501, -64.541, -2.023]
  MoveC 901 to (-345.98, -237.16, -8.16) mm, rotated rx -180 ry 0 rz 0 deg; joints [4.968, -38.054, 103.333, 5.501, -64.509, -2.025] to (-346.16, -237.16, -7.72) mm, rotated rx -180 ry 0 rz 0 deg; joints [4.968, -38.071, 103.321, 5.501, -64.48, -2.028]
  Set speed (1000.0 mm/s)
  MoveL 902 to (-346.16, -237.15, 6) mm, rotated rx -180 ry 0 rz 0 deg; joints [4.965, -38.821, 103.473, 5.525, -63.884, -2.091]
  MoveL 903 to (-219.16, -235.89, 6) mm, rotated rx 180 ry 0 rz 0 deg; joints [5.477, -43.518, 114.711, 5.81, -70.413, -1.598]
  Set speed (25.4 mm/s)
  MoveL 904 to (-219.16, -235.88, -3.54) mm, rotated rx -180 ry 0 rz 0 deg; joints [5.48, -42.939, 114.604, 5.796, -70.882, -1.548]
  MoveC 905 to (-218.98, -235.88, -3.99) mm, rotated rx -180 ry 0 rz 0 deg; joints [5.481, -42.918, 114.615, 5.796, -70.914, -1.545] to (-218.53, -235.89, -4.17) mm, rotated rx 180 ry 0 rz 0 deg; joints [5.483, -42.922, 114.651, 5.796, -70.946, -1.542]
  Set speed (50.8 mm/s)
  MoveL 906 to (-217.89, -235.88, -4.17) mm, rotated rx -180 ry 0 rz 0 deg; joints [5.485, -42.944, 114.704, 5.798, -70.978, -1.54]
  MoveC 907 to (-217.44, -236.07, -4.17) mm, rotated rx -180 ry 0 rz 0 deg; joints [5.479, -42.959, 114.744, 5.791, -71.002, -1.535] to (-217.26, -236.52, -4.17) mm, rotated rx 180 ry 0 rz 0 deg; joints [5.461, -42.967, 114.763, 5.771, -71.013, -1.528]
  MoveL 908 to (-217.26, -261.92, -4.17) mm, rotated rx -180 ry 0 rz 0 deg; joints [4.399, -43.031, 114.947, 4.645, -71.102, -1.168]
  MoveL 909 to (-268.06, -261.92, -4.17) mm, rotated rx -180 ry 0 rz 0 deg; joints [4.241, -41.266, 110.569, 4.554, -68.493, -1.336]
  MoveL 910 to (-268.06, -211.12, -4.18) mm, rotated rx 180 ry 0 rz 0 deg; joints [6.287, -41.116, 110.163, 6.763, -68.31, -2.142]
  MoveL 911 to (-217.26, -211.12, -4.17) mm, rotated rx -180 ry 0 rz 0 deg; joints [6.52, -42.887, 114.539, 6.896, -70.906, -1.894]
  MoveL 912 to (-217.26, -236.52, -4.17) mm, rotated rx 180 ry 0 rz 0 deg; joints [5.461, -42.967, 114.763, 5.771, -71.013, -1.528]
  MoveC 913 to (-217.44, -236.97, -4.17) mm, rotated rx -180 ry 0 rz 0 deg; joints [5.442, -42.962, 114.751, 5.751, -71.005, -1.522] to (-217.89, -237.15, -4.17) mm, rotated rx -180 ry 0 rz 0 deg; joints [5.432, -42.947, 114.715, 5.742, -70.983, -1.522]
  MoveL 914 to (-218.53, -237.16, -4.18) mm, rotated rx 180 ry 0 rz 0 deg; joints [5.43, -42.926, 114.661, 5.74, -70.951, -1.524]
  MoveC 915 to (-218.98, -237.16, -3.99) mm, rotated rx 180 ry 0 rz 0 deg; joints [5.428, -42.922, 114.625, 5.739, -70.919, -1.527] to (-219.16, -237.16, -3.54) mm, rotated rx 180 ry 0 rz 0 deg; joints [5.427, -42.943, 114.614, 5.74, -70.887, -1.53]
  Set speed (1000.0 mm/s)
  MoveL 916 to (-219.16, -237.15, 5) mm, rotated rx 180 ry 0 rz 0 deg; joints [5.425, -43.461, 114.71, 5.752, -70.467, -1.574]
  MoveL 917 to (-219.16, -235.89, 5) mm, rotated rx 180 ry 0 rz 0 deg; joints [5.478, -43.458, 114.7, 5.808, -70.462, -1.593]
  Set speed (25.4 mm/s)
  MoveL 918 to (-219.16, -235.89, 1.82) mm, rotated rx -180 ry 0 rz 0 deg; joints [5.478, -43.265, 114.665, 5.804, -70.619, -1.576]
  MoveL 919 to (-219.16, -235.89, -7.71) mm, rotated rx 180 ry 0 rz 0 deg; joints [5.481, -42.685, 114.555, 5.79, -71.086, -1.527]
  MoveC 920 to (-218.98, -235.88, -8.16) mm, rotated rx -180 ry 0 rz 0 deg; joints [5.482, -42.664, 114.565, 5.79, -71.117, -1.524] to (-218.53, -235.88, -8.35) mm, rotated rx -180 ry 0 rz 0 deg; joints [5.484, -42.668, 114.601, 5.79, -71.149, -1.521]
  Set speed (50.8 mm/s)
  MoveL 921 to (-217.89, -235.88, -8.35) mm, rotated rx -180 ry 0 rz 0 deg; joints [5.486, -42.689, 114.655, 5.792, -71.182, -1.518]
  MoveC 922 to (-217.44, -236.07, -8.35) mm, rotated rx -180 ry 0 rz 0 deg; joints [5.48, -42.705, 114.695, 5.785, -71.206, -1.514] to (-217.26, -236.52, -8.35) mm, rotated rx 180 ry 0 rz 0 deg; joints [5.462, -42.712, 114.714, 5.765, -71.217, -1.507]
  MoveL 923 to (-217.26, -261.92, -8.35) mm, rotated rx -180 ry 0 rz 0 deg; joints [4.4, -42.776, 114.898, 4.64, -71.307, -1.151]
  MoveL 924 to (-268.06, -261.92, -8.35) mm, rotated rx -180 ry 0 rz 0 deg; joints [4.242, -41.022, 110.52, 4.549, -68.688, -1.32]
  MoveL 925 to (-268.06, -211.12, -8.35) mm, rotated rx -180 ry 0 rz 0 deg; joints [6.288, -40.873, 110.114, 6.755, -68.503, -2.117]
  MoveL 926 to (-217.26, -211.12, -8.35) mm, rotated rx -180 ry 0 rz 0 deg; joints [6.521, -42.633, 114.49, 6.889, -71.11, -1.868]
  MoveL 927 to (-217.26, -236.52, -8.35) mm, rotated rx 180 ry 0 rz 0 deg; joints [5.462, -42.712, 114.714, 5.765, -71.217, -1.507]
  MoveC 928 to (-217.44, -236.97, -8.35) mm, rotated rx -180 ry 0 rz 0 deg; joints [5.443, -42.707, 114.702, 5.745, -71.209, -1.501] to (-217.89, -237.16, -8.35) mm, rotated rx 180 ry 0 rz 0 deg; joints [5.433, -42.693, 114.665, 5.736, -71.187, -1.5]
  MoveL 929 to (-218.53, -237.16, -8.35) mm, rotated rx 180 ry 0 rz 0 deg; joints [5.431, -42.672, 114.611, 5.734, -71.154, -1.503]
  MoveC 930 to (-218.98, -237.16, -8.16) mm, rotated rx -180 ry 0 rz 0 deg; joints [5.429, -42.668, 114.575, 5.733, -71.122, -1.506] to (-219.16, -237.16, -7.72) mm, rotated rx 180 ry 0 rz 0 deg; joints [5.428, -42.689, 114.565, 5.734, -71.091, -1.509]
  Set speed (1000.0 mm/s)
  MoveL 931 to (-219.16, -237.15, 6) mm, rotated rx -180 ry 0 rz 0 deg; joints [5.424, -43.522, 114.721, 5.754, -70.417, -1.579]
  MoveL 932 to (-92.16, -235.88, 6) mm, rotated rx -180 ry 0 rz 0 deg; joints [6.036, -47.564, 125.134, 6.197, -76.771, -1.059]
  Set speed (25.4 mm/s)
  MoveL 933 to (-92.16, -235.88, -3.54) mm, rotated rx -180 ry 0 rz 0 deg; joints [6.039, -46.91, 125.02, 6.186, -77.307, -1]
  MoveC 934 to (-91.98, -235.88, -3.99) mm, rotated rx -180 ry 0 rz 0 deg; joints [6.04, -46.885, 125.029, 6.186, -77.342, -0.996] to (-91.53, -235.89, -4.17) mm, rotated rx -180 ry 0 rz 0 deg; joints [6.042, -46.885, 125.063, 6.188, -77.375, -0.993]
  Set speed (50.8 mm/s)
  MoveL 935 to (-90.89, -235.88, -4.18) mm, rotated rx -180 ry 0 rz 0 deg; joints [6.045, -46.903, 125.113, 6.19, -77.407, -0.99]
  MoveC 936 to (-90.44, -236.07, -4.18) mm, rotated rx 180 ry 0 rz 0 deg; joints [6.039, -46.916, 125.15, 6.183, -77.431, -0.986] to (-90.26, -236.52, -4.17) mm, rotated rx 180 ry 0 rz 0 deg; joints [6.019, -46.923, 125.169, 6.163, -77.442, -0.981]
  MoveL 937 to (-90.26, -261.92, -4.18) mm, rotated rx 180 ry 0 rz 0 deg; joints [4.849, -46.981, 125.358, 4.962, -77.55, -0.726]
  MoveL 938 to (-141.06, -261.92, -4.17) mm, rotated rx -180 ry 0 rz 0 deg; joints [4.659, -45.481, 121.277, 4.819, -74.974, -0.909]
  MoveL 939 to (-141.06, -211.12, -4.18) mm, rotated rx -180 ry 0 rz 0 deg; joints [6.903, -45.344, 120.862, 7.151, -74.756, -1.512]
  MoveL 940 to (-90.26, -211.12, -4.18) mm, rotated rx 180 ry 0 rz 0 deg; joints [7.184, -46.85, 124.938, 7.36, -77.313, -1.243]
  MoveL 941 to (-90.26, -236.52, -4.17) mm, rotated rx 180 ry 0 rz 0 deg; joints [6.019, -46.923, 125.169, 6.163, -77.442, -0.981]
  MoveC 942 to (-90.44, -236.97, -4.17) mm, rotated rx -180 ry 0 rz 0 deg; joints [5.998, -46.919, 125.158, 6.141, -77.435, -0.977] to (-90.89, -237.16, -4.17) mm, rotated rx -180 ry 0 rz 0 deg; joints [5.987, -46.906, 125.124, 6.13, -77.413, -0.977]
  MoveL 943 to (-91.53, -237.15, -4.18) mm, rotated rx -180 ry 0 rz 0 deg; joints [5.984, -46.888, 125.073, 6.128, -77.381, -0.98]
  MoveC 944 to (-91.98, -237.15, -3.99) mm, rotated rx -180 ry 0 rz 0 deg; joints [5.982, -46.888, 125.04, 6.126, -77.348, -0.983] to (-92.16, -237.15, -3.54) mm, rotated rx -180 ry 0 rz 0 deg; joints [5.981, -46.914, 125.031, 6.126, -77.313, -0.987]
  Set speed (1000.0 mm/s)
  MoveL 945 to (-92.16, -237.15, 5) mm, rotated rx -180 ry 0 rz 0 deg; joints [5.978, -47.499, 125.133, 6.135, -76.834, -1.039]
  MoveL 946 to (-92.16, -235.88, 5) mm, rotated rx -180 ry 0 rz 0 deg; joints [6.037, -47.495, 125.123, 6.195, -76.828, -1.053]
  Set speed (25.4 mm/s)
  MoveL 947 to (-92.16, -235.88, 1.82) mm, rotated rx -180 ry 0 rz 0 deg; joints [6.038, -47.278, 125.085, 6.192, -77.007, -1.033]
  MoveL 948 to (-92.16, -235.88, -7.71) mm, rotated rx 180 ry 0 rz 0 deg; joints [6.04, -46.624, 124.968, 6.182, -77.54, -0.974]
  MoveC 949 to (-91.98, -235.89, -8.16) mm, rotated rx 180 ry 0 rz 0 deg; joints [6.041, -46.598, 124.977, 6.182, -77.574, -0.971] to (-91.53, -235.88, -8.35) mm, rotated rx -180 ry 0 rz 0 deg; joints [6.044, -46.598, 125.01, 6.183, -77.608, -0.968]
  Set speed (50.8 mm/s)
  MoveL 950 to (-90.89, -235.89, -8.35) mm, rotated rx 180 ry 0 rz 0 deg; joints [6.047, -46.616, 125.06, 6.186, -77.64, -0.965]
  MoveC 951 to (-90.44, -236.07, -8.35) mm, rotated rx -180 ry 0 rz 0 deg; joints [6.04, -46.629, 125.097, 6.179, -77.664, -0.961] to (-90.26, -236.52, -8.35) mm, rotated rx -180 ry 0 rz 0 deg; joints [6.021, -46.636, 125.116, 6.158, -77.675, -0.955]
  MoveL 952 to (-90.26, -261.92, -8.35) mm, rotated rx -180 ry 0 rz 0 deg; joints [4.851, -46.693, 125.305, 4.958, -77.784, -0.706]
  MoveL 953 to (-141.06, -261.92, -8.35) mm, rotated rx 180 ry 0 rz 0 deg; joints [4.66, -45.207, 121.225, 4.815, -75.196, -0.89]
  MoveL 954 to (-141.06, -211.12, -8.35) mm, rotated rx -180 ry 0 rz 0 deg; joints [6.904, -45.072, 120.811, 7.145, -74.976, -1.484]
  MoveL 955 to (-90.26, -211.12, -8.35) mm, rotated rx -180 ry 0 rz 0 deg; joints [7.186, -46.564, 124.885, 7.355, -77.545, -1.213]
  MoveL 956 to (-90.26, -236.52, -8.35) mm, rotated rx -180 ry 0 rz 0 deg; joints [6.021, -46.636, 125.116, 6.158, -77.675, -0.955]
  MoveC 957 to (-90.44, -236.97, -8.35) mm, rotated rx -180 ry 0 rz 0 deg; joints [5.999, -46.632, 125.105, 6.136, -77.668, -0.952] to (-90.89, -237.16, -8.35) mm, rotated rx 180 ry 0 rz 0 deg; joints [5.988, -46.619, 125.071, 6.126, -77.646, -0.952]
  MoveL 958 to (-91.53, -237.15, -8.35) mm, rotated rx -180 ry 0 rz 0 deg; joints [5.985, -46.601, 125.02, 6.124, -77.614, -0.955]
  MoveC 959 to (-91.98, -237.15, -8.16) mm, rotated rx 180 ry 0 rz 0 deg; joints [5.983, -46.601, 124.987, 6.122, -77.58, -0.958] to (-92.16, -237.15, -7.72) mm, rotated rx -180 ry 0 rz 0 deg; joints [5.982, -46.627, 124.978, 6.122, -77.546, -0.962]
  Set speed (1000.0 mm/s)
  MoveL 960 to (-92.16, -237.15, 6) mm, rotated rx -180 ry 0 rz 0 deg; joints [5.978, -47.567, 125.145, 6.137, -76.777, -1.045]
  MoveL 961 to (-92.16, -54.85, 6) mm, rotated rx -180 ry 0 rz 0 deg; joints [14.163, -46.694, 122.589, 14.636, -75.464, -3.259]
  Set speed (25.4 mm/s)
  MoveL 962 to (-92.16, -54.85, -3.54) mm, rotated rx 180 ry 0 rz 0 deg; joints [14.167, -46.062, 122.477, 14.606, -75.968, -3.124]
  MoveC 963 to (-91.98, -54.85, -3.99) mm, rotated rx -180 ry 0 rz 0 deg; joints [14.169, -46.037, 122.486, 14.606, -76.001, -3.115] to (-91.53, -54.85, -4.17) mm, rotated rx -180 ry 0 rz 0 deg; joints [14.174, -46.038, 122.519, 14.609, -76.032, -3.108]
  Set speed (50.8 mm/s)
  MoveL 964 to (-90.89, -54.85, -4.17) mm, rotated rx 180 ry 0 rz 0 deg; joints [14.181, -46.057, 122.569, 14.615, -76.063, -3.102]
  MoveC 965 to (-90.44, -55.04, -4.18) mm, rotated rx 180 ry 0 rz 0 deg; joints [14.178, -46.071, 122.608, 14.61, -76.086, -3.095] to (-90.26, -55.49, -4.17) mm, rotated rx -180 ry 0 rz 0 deg; joints [14.16, -46.08, 122.632, 14.591, -76.1, -3.087]
  MoveL 966 to (-90.26, -80.89, -4.18) mm, rotated rx -180 ry 0 rz 0 deg; joints [13.045, -46.244, 123.112, 13.426, -76.344, -2.752]
  MoveL 967 to (-141.06, -80.89, -4.18) mm, rotated rx 180 ry 0 rz 0 deg; joints [12.546, -44.714, 119.062, 13.063, -73.862, -3.224]
  MoveL 968 to (-141.06, -30.09, -4.17) mm, rotated rx 180 ry 0 rz 0 deg; joints [14.687, -44.357, 118.073, 15.336, -73.395, -3.981]
  MoveL 969 to (-90.26, -30.09, -4.17) mm, rotated rx -180 ry 0 rz 0 deg; joints [15.265, -45.899, 122.111, 15.749, -75.84, -3.437]
  MoveL 970 to (-90.26, -55.49, -4.17) mm, rotated rx -180 ry 0 rz 0 deg; joints [14.16, -46.08, 122.632, 14.591, -76.1, -3.087]
  MoveC 971 to (-90.44, -55.94, -4.18) mm, rotated rx -180 ry 0 rz 0 deg; joints [14.139, -46.077, 122.626, 14.569, -76.095, -3.083] to (-90.89, -56.12, -4.17) mm, rotated rx -180 ry 0 rz 0 deg; joints [14.126, -46.065, 122.594, 14.557, -76.075, -3.085]
  MoveL 972 to (-91.53, -56.12, -4.18) mm, rotated rx 180 ry 0 rz 0 deg; joints [14.119, -46.047, 122.544, 14.551, -76.045, -3.091]
  MoveC 973 to (-91.98, -56.12, -3.99) mm, rotated rx -180 ry 0 rz 0 deg; joints [14.114, -46.046, 122.511, 14.548, -76.013, -3.098] to (-92.16, -56.12, -3.54) mm, rotated rx 180 ry 0 rz 0 deg; joints [14.111, -46.07, 122.502, 14.548, -75.98, -3.106]
  Set speed (1000.0 mm/s)
  MoveL 974 to (-92.16, -56.12, 5) mm, rotated rx 180 ry 0 rz 0 deg; joints [14.108, -46.637, 122.603, 14.575, -75.529, -3.227]
  MoveL 975 to (-92.16, -54.85, 5) mm, rotated rx -180 ry 0 rz 0 deg; joints [14.164, -46.628, 122.578, 14.633, -75.517, -3.244]
  Set speed (25.4 mm/s)
  MoveL 976 to (-92.16, -54.85, 1.83) mm, rotated rx -180 ry 0 rz 0 deg; joints [14.165, -46.418, 122.541, 14.623, -75.685, -3.199]
  MoveL 977 to (-92.16, -54.85, -7.72) mm, rotated rx -180 ry 0 rz 0 deg; joints [14.168, -45.784, 122.426, 14.594, -76.187, -3.065]
  MoveC 978 to (-91.98, -54.85, -8.16) mm, rotated rx -180 ry 0 rz 0 deg; joints [14.171, -45.76, 122.435, 14.594, -76.219, -3.057] to (-91.53, -54.85, -8.35) mm, rotated rx -180 ry 0 rz 0 deg; joints [14.176, -45.76, 122.468, 14.597, -76.251, -3.05]
  Set speed (50.8 mm/s)
  MoveL 979 to (-90.89, -54.85, -8.35) mm, rotated rx -180 ry 0 rz 0 deg; joints [14.183, -45.779, 122.518, 14.602, -76.282, -3.043]
  MoveC 980 to (-90.44, -55.04, -8.35) mm, rotated rx 180 ry 0 rz 0 deg; joints [14.179, -45.793, 122.557, 14.597, -76.305, -3.036] to (-90.26, -55.49, -8.35) mm, rotated rx -180 ry 0 rz 0 deg; joints [14.162, -45.801, 122.58, 14.578, -76.319, -3.028]
  MoveL 981 to (-90.26, -80.89, -8.35) mm, rotated rx -180 ry 0 rz 0 deg; joints [13.047, -45.965, 123.06, 13.415, -76.565, -2.698]
  MoveL 982 to (-141.06, -80.89, -8.35) mm, rotated rx -180 ry 0 rz 0 deg; joints [12.547, -44.448, 119.011, 13.051, -74.073, -3.174]
  MoveL 983 to (-141.06, -30.09, -8.35) mm, rotated rx -180 ry 0 rz 0 deg; joints [14.689, -44.093, 118.023, 15.321, -73.601, -3.923]
  MoveL 984 to (-90.26, -30.09, -8.35) mm, rotated rx 180 ry 0 rz 0 deg; joints [15.266, -45.623, 122.06, 15.735, -76.056, -3.374]
  MoveL 985 to (-90.26, -55.49, -8.35) mm, rotated rx -180 ry 0 rz 0 deg; joints [14.162, -45.801, 122.58, 14.578, -76.319, -3.028]
  MoveC 986 to (-90.44, -55.94, -8.35) mm, rotated rx -180 ry 0 rz 0 deg; joints [14.14, -45.799, 122.574, 14.556, -76.314, -3.024] to (-90.89, -56.12, -8.35) mm, rotated rx -180 ry 0 rz 0 deg; joints [14.127, -45.787, 122.543, 14.544, -76.295, -3.026]
  MoveL 987 to (-91.53, -56.12, -8.35) mm, rotated rx -180 ry 0 rz 0 deg; joints [14.12, -45.769, 122.493, 14.539, -76.264, -3.033]
  MoveC 988 to (-91.98, -56.12, -8.16) mm, rotated rx -180 ry 0 rz 0 deg; joints [14.115, -45.768, 122.46, 14.536, -76.232, -3.04] to (-92.16, -56.12, -7.72) mm, rotated rx 180 ry 0 rz 0 deg; joints [14.113, -45.793, 122.451, 14.536, -76.2, -3.048]
  Set speed (1000.0 mm/s)
  MoveL 989 to (-92.16, -56.12, 6) mm, rotated rx 180 ry 0 rz 0 deg; joints [14.108, -46.703, 122.614, 14.578, -75.476, -3.241]
  MoveL 990 to (-219.16, -54.85, 6) mm, rotated rx -180 ry 0 rz 0 deg; joints [12.889, -42.579, 112.233, 13.787, -69.322, -4.481]
  Set speed (25.4 mm/s)
  MoveL 991 to (-219.16, -54.85, -3.54) mm, rotated rx -180 ry 0 rz 0 deg; joints [12.892, -42.014, 112.128, 13.75, -69.768, -4.366]
  MoveC 992 to (-218.98, -54.85, -3.99) mm, rotated rx 180 ry 0 rz 0 deg; joints [12.894, -41.994, 112.138, 13.749, -69.798, -4.359] to (-218.53, -54.85, -4.17) mm, rotated rx -180 ry 0 rz 0 deg; joints [12.898, -41.999, 112.174, 13.751, -69.829, -4.352]
  Set speed (50.8 mm/s)
  MoveL 993 to (-217.89, -54.85, -4.18) mm, rotated rx -180 ry 0 rz 0 deg; joints [12.904, -42.02, 112.228, 13.754, -69.86, -4.346]
  MoveC 994 to (-217.44, -55.04, -4.18) mm, rotated rx 180 ry 0 rz 0 deg; joints [12.901, -42.037, 112.269, 13.749, -69.884, -4.339] to (-217.26, -55.49, -4.17) mm, rotated rx -180 ry 0 rz 0 deg; joints [12.884, -42.047, 112.294, 13.73, -69.897, -4.329]
  MoveL 995 to (-217.26, -80.89, -4.18) mm, rotated rx -180 ry 0 rz 0 deg; joints [11.863, -42.226, 112.763, 12.623, -70.101, -3.904]
  MoveL 996 to (-268.06, -80.89, -4.17) mm, rotated rx -180 ry 0 rz 0 deg; joints [11.448, -40.434, 108.392, 12.395, -67.552, -4.349]
  MoveL 997 to (-268.06, -30.09, -4.17) mm, rotated rx -180 ry 0 rz 0 deg; joints [13.415, -40.05, 107.417, 14.576, -67.152, -5.286]
  MoveL 998 to (-217.26, -30.09, -4.18) mm, rotated rx -180 ry 0 rz 0 deg; joints [13.897, -41.852, 111.785, 14.834, -69.678, -4.768]
  MoveL 999 to (-217.26, -55.49, -4.17) mm, rotated rx -180 ry 0 rz 0 deg; joints [12.884, -42.047, 112.294, 13.73, -69.897, -4.329]
  MoveC 1000 to (-217.44, -55.94, -4.18) mm, rotated rx -180 ry 0 rz 0 deg; joints [12.865, -42.044, 112.287, 13.71, -69.891, -4.323] to (-217.89, -56.12, -4.18) mm, rotated rx -180 ry 0 rz 0 deg; joints [12.853, -42.03, 112.252, 13.699, -69.871, -4.324]
  MoveL 1001 to (-218.53, -56.12, -4.17) mm, rotated rx -180 ry 0 rz 0 deg; joints [12.847, -42.008, 112.199, 13.696, -69.839, -4.33]
  MoveC 1002 to (-218.98, -56.12, -3.99) mm, rotated rx -180 ry 0 rz 0 deg; joints [12.843, -42.004, 112.163, 13.694, -69.808, -4.337] to (-219.16, -56.12, -3.54) mm, rotated rx -180 ry 0 rz 0 deg; joints [12.841, -42.024, 112.152, 13.695, -69.778, -4.344]
  Set speed (1000.0 mm/s)
  MoveL 1003 to (-219.16, -56.12, 5) mm, rotated rx 180 ry 0 rz 0 deg; joints [12.839, -42.529, 112.247, 13.728, -69.379, -4.447]
  MoveL 1004 to (-219.16, -54.85, 5) mm, rotated rx 180 ry 0 rz 0 deg; joints [12.889, -42.52, 112.223, 13.783, -69.369, -4.469]
  Set speed (25.4 mm/s)
  MoveL 1005 to (-219.16, -54.85, 1.82) mm, rotated rx -180 ry 0 rz 0 deg; joints [12.89, -42.332, 112.188, 13.771, -69.518, -4.43]
  MoveL 1006 to (-219.16, -54.85, -7.71) mm, rotated rx 180 ry 0 rz 0 deg; joints [12.894, -41.767, 112.079, 13.734, -69.961, -4.316]
  MoveC 1007 to (-218.98, -54.85, -8.16) mm, rotated rx -180 ry 0 rz 0 deg; joints [12.895, -41.746, 112.089, 13.734, -69.991, -4.309] to (-218.53, -54.85, -8.35) mm, rotated rx -180 ry 0 rz 0 deg; joints [12.9, -41.751, 112.125, 13.735, -70.022, -4.302]
  Set speed (50.8 mm/s)
  MoveL 1008 to (-217.89, -54.85, -8.35) mm, rotated rx -180 ry 0 rz 0 deg; joints [12.905, -41.772, 112.179, 13.739, -70.054, -4.296]
  MoveC 1009 to (-217.44, -55.04, -8.35) mm, rotated rx 180 ry 0 rz 0 deg; joints [12.902, -41.789, 112.221, 13.733, -70.078, -4.289] to (-217.26, -55.49, -8.35) mm, rotated rx -180 ry 0 rz 0 deg; joints [12.886, -41.799, 112.245, 13.714, -70.091, -4.279]
  MoveL 1010 to (-217.26, -80.89, -8.35) mm, rotated rx 180 ry 0 rz 0 deg; joints [11.865, -41.976, 112.714, 12.608, -70.297, -3.858]
  MoveL 1011 to (-268.06, -80.89, -8.35) mm, rotated rx -180 ry 0 rz 0 deg; joints [11.449, -40.195, 108.344, 12.379, -67.738, -4.305]
  MoveL 1012 to (-268.06, -30.09, -8.35) mm, rotated rx 180 ry 0 rz 0 deg; joints [13.417, -39.813, 107.369, 14.557, -67.335, -5.235]
  MoveL 1013 to (-217.26, -30.09, -8.35) mm, rotated rx -180 ry 0 rz 0 deg; joints [13.899, -41.605, 111.736, 14.817, -69.87, -4.714]
  MoveL 1014 to (-217.26, -55.49, -8.35) mm, rotated rx -180 ry 0 rz 0 deg; joints [12.886, -41.799, 112.245, 13.714, -70.091, -4.279]
  MoveC 1015 to (-217.44, -55.94, -8.35) mm, rotated rx -180 ry 0 rz 0 deg; joints [12.866, -41.796, 112.238, 13.694, -70.085, -4.274] to (-217.89, -56.12, -8.35) mm, rotated rx 180 ry 0 rz 0 deg; joints [12.855, -41.782, 112.203, 13.683, -70.064, -4.275]
  MoveL 1016 to (-218.53, -56.12, -8.35) mm, rotated rx 180 ry 0 rz 0 deg; joints [12.849, -41.76, 112.15, 13.68, -70.033, -4.281]
  MoveC 1017 to (-218.98, -56.12, -8.16) mm, rotated rx -180 ry 0 rz 0 deg; joints [12.845, -41.756, 112.114, 13.678, -70.002, -4.287] to (-219.16, -56.12, -7.72) mm, rotated rx -180 ry 0 rz 0 deg; joints [12.843, -41.776, 112.103, 13.679, -69.972, -4.294]
  Set speed (1000.0 mm/s)
  MoveL 1018 to (-219.16, -56.12, 6) mm, rotated rx -180 ry 0 rz 0 deg; joints [12.838, -42.588, 112.258, 13.732, -69.332, -4.459]
  MoveL 1019 to (-346.16, -54.85, 6) mm, rotated rx -180 ry 0 rz 0 deg; joints [11.822, -37.809, 100.983, 13.297, -62.922, -5.686]
  Set speed (25.4 mm/s)
  MoveL 1020 to (-346.16, -54.85, -3.54) mm, rotated rx -180 ry 0 rz 0 deg; joints [11.825, -37.298, 100.879, 13.252, -63.318, -5.582]
  MoveC 1021 to (-345.98, -54.85, -3.99) mm, rotated rx 180 ry 0 rz 0 deg; joints [11.827, -37.281, 100.892, 13.251, -63.347, -5.576] to (-345.53, -54.85, -4.17) mm, rotated rx -180 ry 0 rz 0 deg; joints [11.83, -37.289, 100.931, 13.251, -63.378, -5.569]
  Set speed (50.8 mm/s)
  MoveL 1022 to (-344.89, -54.85, -4.18) mm, rotated rx -180 ry 0 rz 0 deg; joints [11.835, -37.315, 100.99, 13.253, -63.411, -5.563]
  MoveC 1023 to (-344.44, -55.04, -4.18) mm, rotated rx 180 ry 0 rz 0 deg; joints [11.832, -37.334, 101.036, 13.246, -63.436, -5.555] to (-344.26, -55.49, -4.17) mm, rotated rx -180 ry 0 rz 0 deg; joints [11.817, -37.345, 101.062, 13.227, -63.449, -5.544]
  MoveL 1024 to (-344.26, -80.89, -4.18) mm, rotated rx -180 ry 0 rz 0 deg; joints [10.876, -37.537, 101.532, 12.151, -63.629, -5.024]
  MoveL 1025 to (-395.06, -80.89, -4.18) mm, rotated rx -180 ry 0 rz 0 deg; joints [10.525, -35.452, 96.717, 12.057, -60.926, -5.492]
  MoveL 1026 to (-395.06, -30.09, -4.17) mm, rotated rx 180 ry 0 rz 0 deg; joints [12.343, -35.036, 95.724, 14.202, -60.565, -6.627]
  MoveL 1027 to (-344.26, -30.09, -4.18) mm, rotated rx 180 ry 0 rz 0 deg; joints [12.751, -37.135, 100.551, 14.303, -63.256, -6.076]
  MoveL 1028 to (-344.26, -55.49, -4.17) mm, rotated rx -180 ry 0 rz 0 deg; joints [11.817, -37.345, 101.062, 13.227, -63.449, -5.544]
  MoveC 1029 to (-344.44, -55.94, -4.18) mm, rotated rx 180 ry 0 rz 0 deg; joints [11.799, -37.341, 101.053, 13.208, -63.443, -5.536] to (-344.89, -56.12, -4.17) mm, rotated rx 180 ry 0 rz 0 deg; joints [11.788, -37.325, 101.015, 13.199, -63.42, -5.537]
  MoveL 1030 to (-345.53, -56.12, -4.18) mm, rotated rx -180 ry 0 rz 0 deg; joints [11.783, -37.299, 100.956, 13.197, -63.387, -5.543]
  MoveC 1031 to (-345.98, -56.12, -3.99) mm, rotated rx -180 ry 0 rz 0 deg; joints [11.78, -37.291, 100.916, 13.197, -63.356, -5.549] to (-346.16, -56.12, -3.54) mm, rotated rx 180 ry 0 rz 0 deg; joints [11.778, -37.308, 100.904, 13.199, -63.328, -5.556]
  Set speed (1000.0 mm/s)
  MoveL 1032 to (-346.16, -56.12, 5) mm, rotated rx 180 ry 0 rz 0 deg; joints [11.776, -37.765, 100.997, 13.238, -62.973, -5.648]
  MoveL 1033 to (-346.16, -54.85, 5) mm, rotated rx -180 ry 0 rz 0 deg; joints [11.823, -37.755, 100.972, 13.292, -62.964, -5.675]
  Set speed (25.4 mm/s)
  MoveL 1034 to (-346.16, -54.85, 1.82) mm, rotated rx -180 ry 0 rz 0 deg; joints [11.824, -37.586, 100.938, 13.277, -63.096, -5.64]
  MoveL 1035 to (-346.16, -54.85, -7.72) mm, rotated rx -180 ry 0 rz 0 deg; joints [11.826, -37.074, 100.832, 13.234, -63.491, -5.538]
  MoveC 1036 to (-345.98, -54.85, -8.16) mm, rotated rx -180 ry 0 rz 0 deg; joints [11.828, -37.057, 100.844, 13.232, -63.519, -5.531] to (-345.53, -54.85, -8.35) mm, rotated rx 180 ry 0 rz 0 deg; joints [11.831, -37.065, 100.884, 13.232, -63.55, -5.525]
  Set speed (50.8 mm/s)
  MoveL 1037 to (-344.89, -54.85, -8.35) mm, rotated rx -180 ry 0 rz 0 deg; joints [11.836, -37.09, 100.943, 13.234, -63.583, -5.518]
  MoveC 1038 to (-344.44, -55.04, -8.35) mm, rotated rx -180 ry 0 rz 0 deg; joints [11.833, -37.109, 100.988, 13.227, -63.608, -5.51] to (-344.26, -55.49, -8.35) mm, rotated rx -180 ry 0 rz 0 deg; joints [11.818, -37.12, 101.014, 13.209, -63.621, -5.499]
  MoveL 1039 to (-344.26, -80.89, -8.35) mm, rotated rx 180 ry 0 rz 0 deg; joints [10.877, -37.312, 101.484, 12.134, -63.803, -4.982]
  MoveL 1040 to (-395.06, -80.89, -8.35) mm, rotated rx -180 ry 0 rz 0 deg; joints [10.526, -35.235, 96.669, 12.039, -61.092, -5.452]
  MoveL 1041 to (-395.06, -30.09, -8.35) mm, rotated rx -180 ry 0 rz 0 deg; joints [12.344, -34.82, 95.676, 14.18, -60.728, -6.58]
  MoveL 1042 to (-344.26, -30.09, -8.35) mm, rotated rx -180 ry 0 rz 0 deg; joints [12.752, -36.911, 100.503, 14.283, -63.426, -6.028]
  MoveL 1043 to (-344.26, -55.49, -8.35) mm, rotated rx -180 ry 0 rz 0 deg; joints [11.818, -37.12, 101.014, 13.209, -63.621, -5.499]
  MoveC 1044 to (-344.44, -55.94, -8.35) mm, rotated rx -180 ry 0 rz 0 deg; joints [11.8, -37.117, 101.005, 13.189, -63.615, -5.492] to (-344.89, -56.12, -8.35) mm, rotated rx -180 ry 0 rz 0 deg; joints [11.789, -37.1, 100.967, 13.18, -63.593, -5.492]
  MoveL 1045 to (-345.53, -56.12, -8.35) mm, rotated rx 180 ry 0 rz 0 deg; joints [11.785, -37.075, 100.908, 13.179, -63.56, -5.499]
  MoveC 1046 to (-345.98, -56.12, -8.16) mm, rotated rx -180 ry 0 rz 0 deg; joints [11.781, -37.067, 100.869, 13.178, -63.528, -5.505] to (-346.16, -56.12, -7.72) mm, rotated rx -180 ry 0 rz 0 deg; joints [11.78, -37.084, 100.856, 13.18, -63.5, -5.512]
  Set speed (1000.0 mm/s)
  MoveL 1047 to (-346.16, -56.12, 15) mm, rotated rx -180 ry 0 rz 0 deg; joints [11.773, -38.298, 101.098, 13.286, -62.552, -5.758]
  Print: /'2D Contour1'
  Set speed (1000.0 mm/s)
  MoveL 1048 to (-12.15, 15.92, 15) mm, rotated rx -180 ry 0 rz 0 deg; joints [18.317, -49.068, 127.266, 18.739, -77.936, -3.496]
  MoveL 1049 to (-12.15, 15.92, 6) mm, rotated rx -180 ry 0 rz 0 deg; joints [18.321, -48.437, 127.164, 18.708, -78.437, -3.323]
  Set speed (25.4 mm/s)
  MoveL 1050 to (-12.15, 15.92, -4.37) mm, rotated rx 180 ry 0 rz 0 deg; joints [18.325, -47.709, 127.038, 18.674, -79.009, -3.127]
  MoveC 1051 to (-12.34, 15.92, -4.81) mm, rotated rx -180 ry 0 rz 0 deg; joints [18.323, -47.672, 127.019, 18.67, -79.024, -3.121] to (-12.79, 15.92, -5) mm, rotated rx 180 ry 0 rz 0 deg; joints [18.316, -47.647, 126.983, 18.664, -79.014, -3.123]
  Set speed (50.8 mm/s)
  MoveL 1052 to (-13.42, 15.92, -5) mm, rotated rx -180 ry 0 rz 0 deg; joints [18.307, -47.63, 126.935, 18.656, -78.984, -3.131]
  MoveC 1053 to (-13.87, 16.1, -5) mm, rotated rx -180 ry 0 rz 0 deg; joints [18.308, -47.617, 126.897, 18.66, -78.96, -3.14] to (-14.06, 16.55, -5) mm, rotated rx -180 ry 0 rz 0 deg; joints [18.326, -47.608, 126.872, 18.678, -78.946, -3.148]
  MoveL 1054 to (-14.06, 168.95, -5) mm, rotated rx -180 ry 0 rz 0 deg; joints [24.844, -46.082, 122.399, 25.565, -76.739, -5.587]
  MoveL 1055 to (-39.46, 168.95, -5) mm, rotated rx 180 ry 0 rz 0 deg; joints [24.373, -45.369, 120.514, 25.206, -75.631, -5.996]
  MoveC 1056 to (-52.16, 156.25, -5) mm, rotated rx -180 ry 0 rz 0 deg; joints [23.634, -45.157, 119.983, 24.483, -75.261, -5.955] to (-64.86, 168.95, -5) mm, rotated rx -180 ry 0 rz 0 deg; joints [23.918, -44.631, 118.6, 24.871, -74.514, -6.398]
  MoveL 1057 to (-90.26, 168.95, -5) mm, rotated rx -180 ry 0 rz 0 deg; joints [23.479, -43.869, 116.655, 24.56, -73.387, -6.794]
  MoveL 1058 to (-166.46, 168.95, -5) mm, rotated rx 180 ry 0 rz 0 deg; joints [22.249, -41.435, 110.62, 23.765, -69.937, -7.962]
  MoveC 1059 to (-179.16, 156.25, -5) mm, rotated rx 180 ry 0 rz 0 deg; joints [21.582, -41.171, 109.998, 23.113, -69.513, -7.88] to (-191.86, 168.95, -5) mm, rotated rx -180 ry 0 rz 0 deg; joints [21.866, -40.573, 108.536, 23.544, -68.762, -8.348]
  MoveL 1060 to (-293.46, 168.95, -5) mm, rotated rx 180 ry 0 rz 0 deg; joints [20.452, -36.852, 99.78, 22.89, -63.903, -9.925]
  MoveC 1061 to (-306.16, 156.25, -5) mm, rotated rx 180 ry 0 rz 0 deg; joints [19.844, -36.53, 99.052, 22.3, -63.421, -9.812] to (-318.86, 168.95, -5) mm, rotated rx -180 ry 0 rz 0 deg; joints [20.125, -35.848, 97.471, 22.785, -62.641, -10.335]
  MoveL 1062 to (-395.06, 168.95, -5) mm, rotated rx -180 ry 0 rz 0 deg; joints [19.203, -32.632, 90.194, 22.628, -58.714, -11.639]
  MoveL 1063 to (-420.46, 168.95, -5) mm, rotated rx 180 ry 0 rz 0 deg; joints [18.913, -31.485, 87.635, 22.634, -57.35, -12.107]
  MoveC 1064 to (-433.16, 156.25, -5) mm, rotated rx -180 ry 0 rz 0 deg; joints [18.356, -31.088, 86.766, 22.102, -56.795, -11.977] to (-445.86, 168.95, -5) mm, rotated rx -180 ry 0 rz 0 deg; joints [18.632, -30.294, 84.996, 22.672, -55.952, -12.598]
  MoveL 1065 to (-471.26, 168.95, -5) mm, rotated rx 180 ry 0 rz 0 deg; joints [18.358, -29.057, 82.271, 22.746, -54.518, -13.117]
  MoveL 1066 to (-471.26, 16.55, -5) mm, rotated rx -180 ry 0 rz 0 deg; joints [13.355, -31.1, 86.916, 16.17, -56.002, -8.731]
  MoveL 1067 to (-14.06, 16.55, -5) mm, rotated rx -180 ry 0 rz 0 deg; joints [18.326, -47.608, 126.872, 18.678, -78.946, -3.148]
  MoveC 1068 to (-13.61, 16.36, -5) mm, rotated rx 180 ry 0 rz 0 deg; joints [18.324, -47.622, 126.91, 18.675, -78.969, -3.14] to (-13.42, 15.92, -5) mm, rotated rx -180 ry 0 rz 0 deg; joints [18.307, -47.63, 126.935, 18.656, -78.984, -3.131]
  MoveL 1069 to (-13.42, 15.28, -5) mm, rotated rx 180 ry 0 rz 0 deg; joints [18.278, -47.635, 126.951, 18.627, -78.992, -3.123]
  MoveC 1070 to (-13.42, 14.83, -4.81) mm, rotated rx 180 ry 0 rz 0 deg; joints [18.258, -47.652, 126.964, 18.607, -78.988, -3.12] to (-13.42, 14.65, -4.37) mm, rotated rx 180 ry 0 rz 0 deg; joints [18.25, -47.685, 126.974, 18.599, -78.966, -3.126]
  Set speed (1000.0 mm/s)
  MoveL 1071 to (-13.42, 14.65, 5) mm, rotated rx -180 ry 0 rz 0 deg; joints [18.246, -48.343, 127.089, 18.63, -78.45, -3.303]
  MoveL 1072 to (-12.15, 15.92, 5) mm, rotated rx 180 ry 0 rz 0 deg; joints [18.321, -48.367, 127.153, 18.704, -78.493, -3.304]
  Set speed (25.4 mm/s)
  MoveL 1073 to (-12.15, 15.92, 1) mm, rotated rx -180 ry 0 rz 0 deg; joints [18.323, -48.086, 127.105, 18.691, -78.714, -3.228]
  MoveL 1074 to (-12.15, 15.92, -7.72) mm, rotated rx 180 ry 0 rz 0 deg; joints [18.327, -47.472, 126.996, 18.663, -79.192, -3.064]
  MoveC 1075 to (-12.34, 15.92, -8.16) mm, rotated rx -180 ry 0 rz 0 deg; joints [18.324, -47.436, 126.976, 18.66, -79.207, -3.058] to (-12.79, 15.92, -8.35) mm, rotated rx -180 ry 0 rz 0 deg; joints [18.317, -47.411, 126.94, 18.654, -79.196, -3.061]
  Set speed (50.8 mm/s)
  MoveL 1076 to (-13.42, 15.92, -8.35) mm, rotated rx -180 ry 0 rz 0 deg; joints [18.308, -47.394, 126.892, 18.646, -79.167, -3.069]
  MoveC 1077 to (-13.87, 16.1, -8.35) mm, rotated rx -180 ry 0 rz 0 deg; joints [18.31, -47.381, 126.854, 18.649, -79.143, -3.077] to (-14.06, 16.55, -8.35) mm, rotated rx -180 ry 0 rz 0 deg; joints [18.327, -47.373, 126.829, 18.668, -79.128, -3.086]
  MoveL 1078 to (-14.06, 168.95, -8.35) mm, rotated rx -180 ry 0 rz 0 deg; joints [24.845, -45.86, 122.358, 25.548, -76.902, -5.508]
  MoveL 1079 to (-39.46, 168.95, -8.35) mm, rotated rx 180 ry 0 rz 0 deg; joints [24.374, -45.151, 120.474, 25.189, -75.791, -5.919]
  MoveC 1080 to (-52.16, 156.25, -8.35) mm, rotated rx -180 ry 0 rz 0 deg; joints [23.636, -44.941, 119.943, 24.465, -75.421, -5.881] to (-64.86, 168.95, -8.35) mm, rotated rx -180 ry 0 rz 0 deg; joints [23.919, -44.418, 118.56, 24.853, -74.67, -6.323]
  MoveL 1081 to (-90.26, 168.95, -8.35) mm, rotated rx 180 ry 0 rz 0 deg; joints [23.48, -43.661, 116.615, 24.541, -73.54, -6.722]
  MoveL 1082 to (-166.46, 168.95, -8.35) mm, rotated rx 180 ry 0 rz 0 deg; joints [22.251, -41.239, 110.581, 23.743, -70.081, -7.895]
  MoveC 1083 to (-179.16, 156.25, -8.35) mm, rotated rx 180 ry 0 rz 0 deg; joints [21.583, -40.977, 109.959, 23.091, -69.657, -7.815] to (-191.86, 168.95, -8.35) mm, rotated rx 180 ry 0 rz 0 deg; joints [21.867, -40.381, 108.497, 23.522, -68.903, -8.283]
  MoveL 1084 to (-293.46, 168.95, -8.35) mm, rotated rx 180 ry 0 rz 0 deg; joints [20.453, -36.673, 99.742, 22.865, -64.032, -9.865]
  MoveC 1085 to (-306.16, 156.25, -8.35) mm, rotated rx -180 ry 0 rz 0 deg; joints [19.845, -36.352, 99.014, 22.275, -63.55, -9.754] to (-318.86, 168.95, -8.35) mm, rotated rx -180 ry 0 rz 0 deg; joints [20.126, -35.672, 97.433, 22.759, -62.768, -10.276]
  MoveL 1086 to (-395.06, 168.95, -8.35) mm, rotated rx -180 ry 0 rz 0 deg; joints [19.204, -32.465, 90.156, 22.6, -58.833, -11.582]
  MoveL 1087 to (-420.46, 168.95, -8.35) mm, rotated rx 180 ry 0 rz 0 deg; joints [18.914, -31.32, 87.595, 22.604, -57.466, -12.051]
  MoveC 1088 to (-433.16, 156.25, -8.35) mm, rotated rx 180 ry 0 rz 0 deg; joints [18.357, -30.924, 86.727, 22.073, -56.911, -11.922] to (-445.86, 168.95, -8.35) mm, rotated rx -180 ry 0 rz 0 deg; joints [18.633, -30.132, 84.957, 22.641, -56.066, -12.542]
  MoveL 1089 to (-471.26, 168.95, -8.35) mm, rotated rx 180 ry 0 rz 0 deg; joints [18.359, -28.896, 82.231, 22.715, -54.629, -13.06]
  MoveL 1090 to (-471.26, 16.55, -8.35) mm, rotated rx -180 ry 0 rz 0 deg; joints [13.356, -30.936, 86.876, 16.148, -56.122, -8.69]
  MoveL 1091 to (-14.06, 16.55, -8.35) mm, rotated rx 180 ry 0 rz 0 deg; joints [18.327, -47.373, 126.829, 18.668, -79.128, -3.086]
  MoveC 1092 to (-13.61, 16.36, -8.35) mm, rotated rx -180 ry 0 rz 0 deg; joints [18.325, -47.386, 126.867, 18.665, -79.152, -3.077] to (-13.42, 15.92, -8.35) mm, rotated rx -180 ry 0 rz 0 deg; joints [18.308, -47.394, 126.892, 18.646, -79.167, -3.069]
  MoveL 1093 to (-13.42, 15.28, -8.35) mm, rotated rx -180 ry 0 rz 0 deg; joints [18.28, -47.4, 126.908, 18.616, -79.175, -3.061]
  MoveC 1094 to (-13.42, 14.83, -8.16) mm, rotated rx 180 ry 0 rz 0 deg; joints [18.26, -47.416, 126.921, 18.596, -79.171, -3.058] to (-13.42, 14.65, -7.72) mm, rotated rx -180 ry 0 rz 0 deg; joints [18.251, -47.449, 126.932, 18.589, -79.149, -3.064]
  Set speed (1000.0 mm/s)
  MoveL 1095 to (-13.42, 14.65, 6) mm, rotated rx 180 ry 0 rz 0 deg; joints [18.245, -48.413, 127.1, 18.633, -78.395, -3.322]
  MoveL 1096 to (18.41, 14.65, 6) mm, rotated rx 180 ry 0 rz 0 deg; joints [18.726, -49.26, 129.471, 19.028, -79.865, -2.906]
  Set speed (25.4 mm/s)
  MoveL 1097 to (18.41, 14.65, -4.36) mm, rotated rx -180 ry 0 rz 0 deg; joints [18.731, -48.508, 129.342, 18.997, -80.455, -2.7]
  MoveC 1098 to (18.41, 14.83, -4.81) mm, rotated rx -180 ry 0 rz 0 deg; joints [18.739, -48.474, 129.332, 19.005, -80.478, -2.694] to (18.41, 15.28, -5) mm, rotated rx -180 ry 0 rz 0 deg; joints [18.76, -48.457, 129.318, 19.025, -80.482, -2.696]
  Set speed (50.8 mm/s)
  MoveL 1099 to (18.41, 15.92, -5) mm, rotated rx -180 ry 0 rz 0 deg; joints [18.789, -48.452, 129.302, 19.055, -80.473, -2.704]
  MoveC 1100 to (18.6, 16.36, -5) mm, rotated rx -180 ry 0 rz 0 deg; joints [18.812, -48.453, 129.305, 19.079, -80.476, -2.707] to (19.05, 16.55, -5) mm, rotated rx 180 ry 0 rz 0 deg; joints [18.828, -48.463, 129.333, 19.094, -80.494, -2.703]
  MoveL 1101 to (39.46, 16.55, -5) mm, rotated rx 180 ry 0 rz 0 deg; joints [19.151, -48.966, 130.831, 19.368, -81.448, -2.418]
  MoveL 1102 to (471.26, 16.55, -5) mm, rotated rx 180 ry 0 rz 30 deg; joints [37.52, -54.012, 150.509, 67.557, -91.595, 5.804]
  MoveL 1103 to (471.26, 168.95, -5) mm, rotated rx 180 ry 0 rz 0 deg; joints [38.577, -54.253, 153.452, 38.847, -96.315, 6.028]
  MoveL 1104 to (445.86, 168.95, -5) mm, rotated rx 180 ry 0 rz 0 deg; joints [37.545, -54.152, 152.058, 37.732, -95.395, 5.101]
  MoveC 1105 to (433.16, 156.25, -5) mm, rotated rx -180 ry 0 rz 0 deg; joints [36.387, -54.114, 151.879, 36.564, -95.378, 4.889] to (420.46, 168.95, -5) mm, rotated rx -180 ry 0 rz 0 deg; joints [36.558, -54.006, 150.636, 36.678, -94.455, 4.228]
  MoveL 1106 to (395.06, 168.95, -5) mm, rotated rx -180 ry 0 rz 0 deg; joints [35.616, -53.815, 149.187, 35.683, -93.498, 3.404]
  MoveL 1107 to (318.86, 168.95, -5) mm, rotated rx -180 ry 0 rz 0 deg; joints [33.027, -52.998, 144.685, 33.02, -90.545, 1.191]
  MoveC 1108 to (306.16, 156.25, -5) mm, rotated rx -180 ry 0 rz 0 deg; joints [32.006, -52.921, 144.401, 31.999, -90.386, 1.057] to (293.46, 168.95, -5) mm, rotated rx -180 ry 0 rz 0 deg; joints [32.237, -52.652, 143.134, 32.23, -89.538, 0.529]
  MoveL 1109 to (191.86, 168.95, -5) mm, rotated rx -180 ry 0 rz 0 deg; joints [29.39, -50.937, 136.686, 29.486, -85.428, -1.819]
  MoveC 1110 to (179.16, 156.25, -5) mm, rotated rx -180 ry 0 rz 0 deg; joints [28.486, -50.813, 136.31, 28.589, -85.175, -1.881] to (166.46, 168.95, -5) mm, rotated rx 180 ry 0 rz 0 deg; joints [28.749, -50.432, 135.013, 28.893, -84.382, -2.343]
  MoveL 1111 to (90.26, 168.95, -5) mm, rotated rx -180 ry 0 rz 0 deg; joints [26.97, -48.754, 129.848, 27.311, -81.201, -3.802]
  MoveL 1112 to (64.86, 168.95, -5) mm, rotated rx 180 ry 0 rz 0 deg; joints [26.422, -48.143, 128.075, 26.843, -80.127, -4.255]
  MoveC 1113 to (61.14, 159.97, -5) mm, rotated rx -180 ry 0 rz 0 deg; joints [25.96, -48.152, 128.123, 26.373, -80.125, -4.165] to (52.16, 156.25, -5) mm, rotated rx -180 ry 0 rz 0 deg; joints [25.615, -47.97, 127.614, 26.05, -79.804, -4.256]
  MoveL 1114 to (52.16, 156.25, -5) mm, rotated rx -180 ry 0 rz 0 deg; joints [25.615, -47.97, 127.614, 26.05, -79.804, -4.256]
  MoveC 1115 to (43.18, 159.97, -5) mm, rotated rx 180 ry 0 rz 0 deg; joints [25.591, -47.703, 126.849, 26.065, -79.355, -4.474] to (39.46, 168.95, -5) mm, rotated rx -180 ry 0 rz 0 deg; joints [25.894, -47.506, 126.277, 26.404, -79.044, -4.696]
  MoveL 1116 to (14.06, 168.95, -5) mm, rotated rx -180 ry 0 rz 0 deg; joints [25.385, -46.844, 124.451, 25.991, -77.955, -5.125]
  MoveL 1117 to (14.06, 16.55, -5) mm, rotated rx -180 ry 0 rz 0 deg; joints [18.75, -48.337, 128.965, 19.029, -80.261, -2.771]
  MoveL 1118 to (19.05, 16.55, -5) mm, rotated rx 180 ry 0 rz 0 deg; joints [18.828, -48.463, 129.333, 19.094, -80.494, -2.703]
  MoveC 1119 to (19.49, 16.36, -5) mm, rotated rx -180 ry 0 rz 0 deg; joints [18.826, -48.475, 129.371, 19.091, -80.518, -2.695] to (19.68, 15.92, -5) mm, rotated rx -180 ry 0 rz 0 deg; joints [18.809, -48.483, 129.396, 19.072, -80.533, -2.686]
  MoveL 1120 to (19.68, 15.28, -5) mm, rotated rx -180 ry 0 rz 0 deg; joints [18.78, -48.488, 129.412, 19.042, -80.542, -2.678]
  MoveC 1121 to (19.68, 14.83, -4.81) mm, rotated rx -180 ry 0 rz 0 deg; joints [18.759, -48.505, 129.425, 19.021, -80.537, -2.676] to (19.68, 14.65, -4.37) mm, rotated rx -180 ry 0 rz 0 deg; joints [18.75, -48.54, 129.436, 19.014, -80.514, -2.683]
  Set speed (1000.0 mm/s)
  MoveL 1122 to (19.68, 14.65, 5) mm, rotated rx -180 ry 0 rz 0 deg; joints [18.746, -49.22, 129.553, 19.041, -79.981, -2.869]
  MoveL 1123 to (18.41, 14.65, 5) mm, rotated rx -180 ry 0 rz 0 deg; joints [18.726, -49.187, 129.459, 19.025, -79.923, -2.886]
  Set speed (25.4 mm/s)
  MoveL 1124 to (18.41, 14.65, 1) mm, rotated rx -180 ry 0 rz 0 deg; joints [18.728, -48.897, 129.41, 19.013, -80.151, -2.806]
  MoveL 1125 to (18.41, 14.65, -7.71) mm, rotated rx -180 ry 0 rz 0 deg; joints [18.732, -48.264, 129.298, 18.988, -80.644, -2.635]
  MoveC 1126 to (18.41, 14.83, -8.16) mm, rotated rx 180 ry 0 rz 0 deg; joints [18.741, -48.23, 129.288, 18.995, -80.667, -2.628] to (18.41, 15.28, -8.35) mm, rotated rx -180 ry 0 rz 0 deg; joints [18.761, -48.213, 129.274, 19.016, -80.671, -2.63]
  Set speed (50.8 mm/s)
  MoveL 1127 to (18.41, 15.92, -8.35) mm, rotated rx -180 ry 0 rz 0 deg; joints [18.79, -48.208, 129.258, 19.046, -80.662, -2.638]
  MoveC 1128 to (18.6, 16.36, -8.35) mm, rotated rx 180 ry 0 rz 0 deg; joints [18.814, -48.209, 129.261, 19.07, -80.665, -2.641] to (19.04, 16.55, -8.35) mm, rotated rx -180 ry 0 rz 0 deg; joints [18.829, -48.219, 129.289, 19.084, -80.683, -2.637]
  MoveL 1129 to (39.46, 16.55, -8.35) mm, rotated rx -180 ry 0 rz 0 deg; joints [19.153, -48.717, 130.786, 19.36, -81.641, -2.35]
  MoveL 1130 to (471.26, 16.55, -8.35) mm, rotated rx 180 ry 0 rz 30 deg; joints [37.523, -53.659, 150.449, 67.567, -91.707, 6.076]
  MoveL 1131 to (471.26, 168.95, -8.35) mm, rotated rx 180 ry 0 rz 0 deg; joints [38.58, -53.874, 153.388, 38.873, -96.56, 6.227]
  MoveL 1132 to (445.86, 168.95, -8.35) mm, rotated rx 180 ry 0 rz 0 deg; joints [37.547, -53.786, 151.996, 37.752, -95.636, 5.289]
  MoveC 1133 to (433.16, 156.25, -8.35) mm, rotated rx -180 ry 0 rz 0 deg; joints [36.389, -53.749, 151.817, 36.585, -95.621, 5.071] to (420.46, 168.95, -8.35) mm, rotated rx 180 ry 0 rz 0 deg; joints [36.561, -53.651, 150.577, 36.695, -94.691, 4.405]
  MoveL 1134 to (395.06, 168.95, -8.35) mm, rotated rx -180 ry 0 rz 0 deg; joints [35.618, -53.471, 149.129, 35.696, -93.73, 3.571]
  MoveL 1135 to (318.86, 168.95, -8.35) mm, rotated rx 180 ry 0 rz 0 deg; joints [33.029, -52.685, 144.631, 33.024, -90.763, 1.333]
  MoveC 1136 to (306.16, 156.25, -8.35) mm, rotated rx -180 ry 0 rz 0 deg; joints [32.009, -52.609, 144.348, 32.002, -90.605, 1.194] to (293.46, 168.95, -8.35) mm, rotated rx -180 ry 0 rz 0 deg; joints [32.239, -52.347, 143.082, 32.231, -89.752, 0.664]
  MoveL 1137 to (191.86, 168.95, -8.35) mm, rotated rx 180 ry 0 rz 0 deg; joints [29.392, -50.665, 136.638, 29.479, -85.624, -1.708]
  MoveC 1138 to (179.16, 156.25, -8.35) mm, rotated rx 180 ry 0 rz 0 deg; joints [28.488, -50.542, 136.263, 28.582, -85.371, -1.774] to (166.46, 168.95, -8.35) mm, rotated rx 180 ry 0 rz 0 deg; joints [28.751, -50.167, 134.967, 28.885, -84.573, -2.237]
  MoveL 1139 to (90.26, 168.95, -8.35) mm, rotated rx -180 ry 0 rz 0 deg; joints [26.972, -48.509, 129.804, 27.298, -81.38, -3.708]
  MoveL 1140 to (64.86, 168.95, -8.35) mm, rotated rx 180 ry 0 rz 0 deg; joints [26.424, -47.903, 128.032, 26.83, -80.302, -4.166]
  MoveC 1141 to (61.14, 159.97, -8.35) mm, rotated rx 180 ry 0 rz 0 deg; joints [25.962, -47.912, 128.08, 26.36, -80.301, -4.077] to (52.16, 156.25, -8.35) mm, rotated rx -180 ry 0 rz 0 deg; joints [25.617, -47.733, 127.571, 26.036, -79.979, -4.17]
  MoveL 1142 to (52.16, 156.25, -8.35) mm, rotated rx -180 ry 0 rz 0 deg; joints [25.617, -47.733, 127.571, 26.036, -79.979, -4.17]
  MoveC 1143 to (43.18, 159.97, -8.35) mm, rotated rx -180 ry 0 rz 0 deg; joints [25.592, -47.467, 126.807, 26.051, -79.529, -4.388] to (39.46, 168.95, -8.35) mm, rotated rx -180 ry 0 rz 0 deg; joints [25.896, -47.272, 126.234, 26.389, -79.216, -4.61]
  MoveL 1144 to (14.06, 168.95, -8.35) mm, rotated rx 180 ry 0 rz 0 deg; joints [25.387, -46.615, 124.41, 25.976, -78.122, -5.042]
  MoveL 1145 to (14.06, 16.55, -8.35) mm, rotated rx 180 ry 0 rz 0 deg; joints [18.752, -48.094, 128.921, 19.019, -80.449, -2.706]
  MoveL 1146 to (19.04, 16.55, -8.35) mm, rotated rx -180 ry 0 rz 0 deg; joints [18.829, -48.219, 129.289, 19.084, -80.683, -2.637]
  MoveC 1147 to (19.49, 16.36, -8.35) mm, rotated rx -180 ry 0 rz 0 deg; joints [18.828, -48.232, 129.327, 19.081, -80.707, -2.629] to (19.68, 15.92, -8.35) mm, rotated rx -180 ry 0 rz 0 deg; joints [18.81, -48.24, 129.352, 19.063, -80.722, -2.62]
  MoveL 1148 to (19.68, 15.28, -8.35) mm, rotated rx -180 ry 0 rz 0 deg; joints [18.781, -48.245, 129.368, 19.033, -80.731, -2.612]
  MoveC 1149 to (19.68, 14.83, -8.16) mm, rotated rx -180 ry 0 rz 0 deg; joints [18.761, -48.262, 129.381, 19.012, -80.726, -2.611] to (19.68, 14.65, -7.72) mm, rotated rx -180 ry 0 rz 0 deg; joints [18.752, -48.296, 129.392, 19.004, -80.704, -2.617]
  Set speed (1000.0 mm/s)
  MoveL 1150 to (19.68, 14.65, 6) mm, rotated rx -180 ry 0 rz 0 deg; joints [18.746, -49.293, 129.565, 19.044, -79.924, -2.889]
  MoveL 1151 to (12.15, -16.75, 6) mm, rotated rx -180 ry 0 rz 0 deg; joints [17.189, -49.34, 129.757, 17.457, -79.981, -2.59]
  Set speed (25.4 mm/s)
  MoveL 1152 to (12.15, -16.75, -4.36) mm, rotated rx 180 ry 0 rz 0 deg; joints [17.193, -48.584, 129.628, 17.43, -80.578, -2.401]
  MoveC 1153 to (12.34, -16.75, -4.81) mm, rotated rx 180 ry 0 rz 0 deg; joints [17.196, -48.556, 129.636, 17.431, -80.613, -2.39] to (12.79, -16.75, -5) mm, rotated rx -180 ry 0 rz 0 deg; joints [17.203, -48.554, 129.667, 17.436, -80.645, -2.381]
  Set speed (50.8 mm/s)
  MoveL 1154 to (13.42, -16.75, -5) mm, rotated rx 180 ry 0 rz 0 deg; joints [17.212, -48.57, 129.714, 17.443, -80.675, -2.373]
  MoveC 1155 to (13.87, -16.94, -5) mm, rotated rx -180 ry 0 rz 0 deg; joints [17.21, -48.582, 129.752, 17.44, -80.699, -2.365] to (14.06, -17.39, -5) mm, rotated rx -180 ry 0 rz 0 deg; joints [17.191, -48.59, 129.776, 17.421, -80.714, -2.357]
  MoveL 1156 to (14.06, -169.79, -5) mm, rotated rx 180 ry 0 rz 0 deg; joints [9.889, -49.4, 132.515, 9.973, -82.348, -0.917]
  MoveL 1157 to (471.26, -169.79, -5) mm, rotated rx 180 ry 0 rz 30 deg; joints [26.888, -53.923, 157.36, 57.435, -96.421, 11.096]
  MoveL 1158 to (471.26, -17.39, -5) mm, rotated rx -180 ry 0 rz 30 deg; joints [35.768, -54.104, 151.92, 65.857, -92.317, 6.931]
  MoveL 1159 to (445.86, -17.39, -5) mm, rotated rx -180 ry 0 rz 30 deg; joints [34.824, -53.952, 150.466, 64.875, -91.882, 5.697]
